Yaskawa INFORM job: A_ROOF_UPPER_0614_2_PAINT_31.JBI

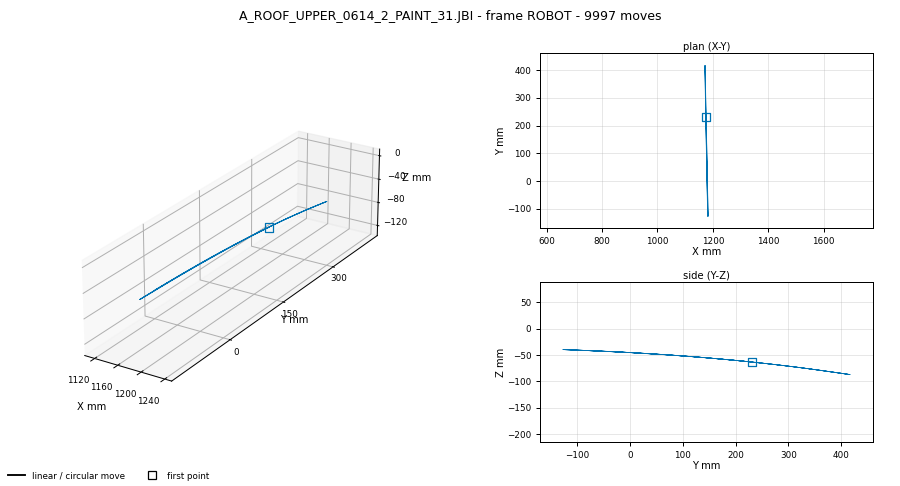
[picture p0: tool path of A_ROOF_UPPER_0614_2_PAINT_31.JBI in frame ROBOT, 9997 of 9997 moves have a stored position in this frame; points joined in program order, loops and branches not executed]
/JOB
//NAME A_ROOF_UPPER_0614_2_PAINT31
//POS
///NPOS 9997,0,0,0,0,0
///TOOL 1
///USER 0
///POSTYPE ROBOT
///RECTAN
///RCONF 1,0,0,0,0,0,0,0,0,0,0,0,0,0,0,0,0,0,0,0,0,0,0,0
C00000=1175.962,231.561,-63.142,-177.522,7.133,148.611
C00001=1175.967,231.312,-63.116,-177.525,7.130,148.612
C00002=1175.971,231.063,-63.091,-177.528,7.128,148.612
C00003=1175.976,230.815,-63.065,-177.530,7.126,148.612
C00004=1175.980,230.567,-63.040,-177.533,7.123,148.612
C00005=1175.985,230.317,-63.013,-177.535,7.121,148.612
C00006=1175.989,230.069,-62.987,-177.539,7.118,148.613
C00007=1175.994,229.820,-62.962,-177.541,7.116,148.613
C00008=1175.998,229.572,-62.936,-177.544,7.113,148.613
C00009=1176.002,229.323,-62.911,-177.546,7.111,148.613
C00010=1176.007,229.075,-62.885,-177.550,7.109,148.614
C00011=1176.011,228.826,-62.859,-177.552,7.107,148.614
C00012=1176.016,228.577,-62.834,-177.555,7.104,148.614
C00013=1176.020,228.328,-62.808,-177.557,7.102,148.614
C00014=1176.025,228.080,-62.783,-177.560,7.099,148.614
C00015=1176.030,227.831,-62.756,-177.563,7.097,148.614
C00016=1176.034,227.582,-62.730,-177.565,7.094,148.615
C00017=1176.039,227.334,-62.705,-177.568,7.092,148.615
C00018=1176.043,227.085,-62.679,-177.571,7.089,148.615
C00019=1176.047,226.837,-62.654,-177.573,7.087,148.615
C00020=1176.052,226.589,-62.628,-177.576,7.085,148.615
C00021=1176.057,226.339,-62.603,-177.579,7.083,148.616
C00022=1176.061,226.091,-62.578,-177.581,7.081,148.616
C00023=1176.066,225.842,-62.552,-177.584,7.078,148.616
C00024=1176.070,225.593,-62.526,-177.586,7.076,148.616
C00025=1176.075,225.345,-62.501,-177.590,7.073,148.616
C00026=1176.079,225.096,-62.476,-177.592,7.071,148.617
C00027=1176.083,224.847,-62.450,-177.595,7.068,148.617
C00028=1176.088,224.599,-62.425,-177.597,7.066,148.617
C00029=1176.092,224.350,-62.400,-177.600,7.065,148.617
C00030=1176.097,224.102,-62.375,-177.603,7.062,148.618
C00031=1176.101,223.853,-62.349,-177.605,7.060,148.618
C00032=1176.105,223.604,-62.323,-177.608,7.057,148.618
C00033=1176.110,223.356,-62.298,-177.611,7.055,148.618
C00034=1176.115,223.107,-62.273,-177.614,7.052,148.618
C00035=1176.119,222.858,-62.248,-177.616,7.050,148.619
C00036=1176.124,222.610,-62.222,-177.619,7.048,148.619
C00037=1176.129,222.361,-62.197,-177.621,7.045,148.619
C00038=1176.133,222.112,-62.171,-177.624,7.044,148.619
C00039=1176.137,221.863,-62.146,-177.627,7.041,148.619
C00040=1176.142,221.615,-62.122,-177.630,7.039,148.620
C00041=1176.146,221.366,-62.096,-177.632,7.036,148.620
C00042=1176.151,221.117,-62.071,-177.635,7.034,148.620
C00043=1176.155,220.869,-62.045,-177.637,7.032,148.620
C00044=1176.160,220.620,-62.020,-177.640,7.029,148.621
C00045=1176.165,220.371,-61.995,-177.643,7.028,148.621
C00046=1176.169,220.123,-61.970,-177.646,7.025,148.621
C00047=1176.173,219.874,-61.945,-177.648,7.023,148.621
C00048=1176.178,219.626,-61.920,-177.651,7.021,148.621
C00049=1176.183,219.376,-61.895,-177.654,7.018,148.622
C00050=1176.187,219.129,-61.870,-177.656,7.016,148.622
C00051=1176.191,218.879,-61.845,-177.659,7.013,148.622
C00052=1176.196,218.631,-61.820,-177.662,7.012,148.623
C00053=1176.201,218.382,-61.795,-177.664,7.009,148.623
C00054=1176.205,218.134,-61.770,-177.667,7.007,148.623
C00055=1176.209,217.884,-61.745,-177.670,7.005,148.623
C00056=1176.214,217.636,-61.720,-177.673,7.002,148.623
C00057=1176.219,217.387,-61.694,-177.675,7.000,148.623
C00058=1176.223,217.138,-61.670,-177.678,6.998,148.624
C00059=1176.227,216.890,-61.644,-177.681,6.996,148.624
C00060=1176.232,216.641,-61.620,-177.683,6.993,148.624
C00061=1176.236,216.392,-61.595,-177.686,6.991,148.625
C00062=1176.241,216.144,-61.570,-177.688,6.989,148.625
C00063=1176.245,215.894,-61.545,-177.691,6.987,148.625
C00064=1176.250,215.646,-61.521,-177.694,6.984,148.625
C00065=1176.255,215.398,-61.495,-177.697,6.982,148.625
C00066=1176.259,215.148,-61.470,-177.699,6.980,148.626
C00067=1176.264,214.900,-61.446,-177.702,6.977,148.626
C00068=1176.268,214.651,-61.421,-177.705,6.976,148.626
C00069=1176.273,214.402,-61.396,-177.708,6.973,148.626
C00070=1176.277,214.153,-61.371,-177.710,6.971,148.627
C00071=1176.282,213.905,-61.347,-177.713,6.969,148.627
C00072=1176.287,213.656,-61.321,-177.715,6.966,148.627
C00073=1176.290,213.407,-61.297,-177.718,6.964,148.627
C00074=1176.296,213.159,-61.272,-177.721,6.962,148.628
C00075=1176.300,212.910,-61.248,-177.724,6.960,148.628
C00076=1176.305,212.661,-61.223,-177.726,6.958,148.628
C00077=1176.309,212.413,-61.198,-177.728,6.956,148.628
C00078=1176.313,212.164,-61.173,-177.732,6.953,148.629
C00079=1176.318,211.915,-61.149,-177.734,6.951,148.629
C00080=1176.323,211.666,-61.125,-177.736,6.949,148.629
C00081=1176.327,211.417,-61.100,-177.740,6.946,148.629
C00082=1176.332,211.169,-61.076,-177.742,6.945,148.630
C00083=1176.337,210.920,-61.051,-177.745,6.942,148.630
C00084=1176.341,210.649,-61.024,-177.748,6.940,148.630
C00085=1176.346,210.379,-60.998,-177.751,6.937,148.630
C00086=1176.351,210.109,-60.971,-177.754,6.935,148.631
C00087=1176.355,209.838,-60.944,-177.756,6.933,148.631
C00088=1176.361,209.589,-60.919,-177.759,6.931,148.631
C00089=1176.365,209.341,-60.895,-177.762,6.928,148.631
C00090=1176.369,209.092,-60.870,-177.765,6.926,148.632
C00091=1176.374,208.843,-60.846,-177.767,6.924,148.632
C00092=1176.379,208.594,-60.821,-177.770,6.922,148.632
C00093=1176.383,208.346,-60.797,-177.773,6.919,148.632
C00094=1176.387,208.097,-60.773,-177.775,6.918,148.633
C00095=1176.392,207.848,-60.748,-177.779,6.915,148.633
C00096=1176.397,207.600,-60.724,-177.781,6.913,148.633
C00097=1176.402,207.351,-60.699,-177.783,6.911,148.634
C00098=1176.406,207.102,-60.675,-177.787,6.909,148.634
C00099=1176.411,206.853,-60.651,-177.789,6.906,148.634
C00100=1176.415,206.604,-60.627,-177.791,6.905,148.634
C00101=1176.420,206.356,-60.603,-177.795,6.902,148.635
C00102=1176.424,206.106,-60.578,-177.797,6.900,148.635
C00103=1176.429,205.858,-60.554,-177.800,6.898,148.635
C00104=1176.433,205.609,-60.530,-177.802,6.896,148.635
C00105=1176.438,205.361,-60.505,-177.805,6.893,148.636
C00106=1176.442,205.111,-60.481,-177.808,6.892,148.636
C00107=1176.447,204.863,-60.457,-177.810,6.890,148.636
C00108=1176.452,204.614,-60.433,-177.813,6.887,148.636
C00109=1176.456,204.365,-60.408,-177.816,6.885,148.637
C00110=1176.461,204.117,-60.384,-177.818,6.883,148.637
C00111=1176.466,203.867,-60.360,-177.821,6.880,148.637
C00112=1176.470,203.619,-60.336,-177.824,6.878,148.637
C00113=1176.474,203.370,-60.312,-177.827,6.877,148.638
C00114=1176.479,203.122,-60.288,-177.829,6.875,148.638
C00115=1176.484,202.872,-60.264,-177.832,6.872,148.638
C00116=1176.488,202.623,-60.239,-177.835,6.870,148.639
C00117=1176.492,202.375,-60.215,-177.837,6.868,148.639
C00118=1176.497,202.126,-60.192,-177.840,6.865,148.639
C00119=1176.502,201.877,-60.167,-177.843,6.864,148.639
C00120=1176.507,201.629,-60.143,-177.845,6.862,148.640
C00121=1176.511,201.380,-60.120,-177.848,6.860,148.640
C00122=1176.515,201.131,-60.096,-177.851,6.857,148.640
C00123=1176.519,200.882,-60.071,-177.853,6.855,148.640
C00124=1176.525,200.633,-60.047,-177.856,6.853,148.641
C00125=1176.529,200.384,-60.023,-177.859,6.851,148.641
C00126=1176.534,200.135,-60.000,-177.862,6.849,148.641
C00127=1176.538,199.887,-59.976,-177.864,6.847,148.642
C00128=1176.543,199.639,-59.952,-177.866,6.845,148.642
C00129=1176.547,199.389,-59.928,-177.870,6.842,148.642
C00130=1176.552,199.140,-59.904,-177.872,6.840,148.642
C00131=1176.557,198.891,-59.880,-177.875,6.839,148.643
C00132=1176.561,198.643,-59.856,-177.877,6.837,148.643
C00133=1176.566,198.394,-59.833,-177.880,6.834,148.643
C00134=1176.570,198.145,-59.809,-177.883,6.832,148.644
C00135=1176.575,197.896,-59.785,-177.885,6.830,148.644
C00136=1176.579,197.648,-59.761,-177.888,6.828,148.644
C00137=1176.584,197.399,-59.738,-177.891,6.826,148.644
C00138=1176.588,197.150,-59.714,-177.894,6.824,148.645
C00139=1176.593,196.901,-59.690,-177.896,6.822,148.645
C00140=1176.598,196.653,-59.666,-177.899,6.820,148.645
C00141=1176.602,196.403,-59.642,-177.902,6.817,148.646
C00142=1176.607,196.154,-59.619,-177.905,6.816,148.646
C00143=1176.611,195.905,-59.595,-177.907,6.813,148.646
C00144=1176.616,195.656,-59.571,-177.910,6.812,148.646
C00145=1176.621,195.407,-59.548,-177.913,6.809,148.647
C00146=1176.625,195.159,-59.524,-177.915,6.807,148.647
C00147=1176.630,194.910,-59.500,-177.918,6.805,148.647
C00148=1176.635,194.661,-59.477,-177.920,6.803,148.648
C00149=1176.639,194.412,-59.453,-177.923,6.802,148.648
C00150=1176.644,194.163,-59.430,-177.926,6.799,148.648
C00151=1176.648,193.914,-59.406,-177.928,6.797,148.648
C00152=1176.653,193.666,-59.382,-177.931,6.795,148.649
C00153=1176.657,193.417,-59.359,-177.934,6.793,148.649
C00154=1176.662,193.168,-59.335,-177.937,6.791,148.649
C00155=1176.667,192.919,-59.312,-177.940,6.789,148.650
C00156=1176.671,192.670,-59.288,-177.942,6.787,148.650
C00157=1176.675,192.422,-59.265,-177.945,6.785,148.650
C00158=1176.680,192.173,-59.242,-177.947,6.783,148.651
C00159=1176.685,191.924,-59.219,-177.950,6.781,148.651
C00160=1176.689,191.675,-59.195,-177.953,6.779,148.651
C00161=1176.694,191.426,-59.171,-177.955,6.777,148.651
C00162=1176.699,191.178,-59.148,-177.958,6.775,148.652
C00163=1176.704,190.929,-59.125,-177.961,6.773,148.652
C00164=1176.708,190.680,-59.101,-177.964,6.771,148.652
C00165=1176.713,190.431,-59.078,-177.966,6.768,148.652
C00166=1176.718,190.182,-59.055,-177.969,6.767,148.653
C00167=1176.721,189.934,-59.031,-177.971,6.765,148.653
C00168=1176.726,189.685,-59.008,-177.974,6.763,148.654
C00169=1176.731,189.436,-58.985,-177.977,6.760,148.654
C00170=1176.736,189.187,-58.961,-177.980,6.758,148.654
C00171=1176.740,188.938,-58.938,-177.982,6.757,148.654
C00172=1176.745,188.688,-58.914,-177.985,6.755,148.655
C00173=1176.749,188.440,-58.892,-177.988,6.753,148.655
C00174=1176.754,188.191,-58.869,-177.991,6.750,148.655
C00175=1176.759,187.942,-58.845,-177.993,6.748,148.656
C00176=1176.764,187.693,-58.822,-177.996,6.747,148.656
C00177=1176.768,187.444,-58.799,-177.998,6.745,148.656
C00178=1176.772,187.196,-58.776,-178.001,6.743,148.657
C00179=1176.777,186.947,-58.752,-178.004,6.741,148.657
C00180=1176.782,186.698,-58.729,-178.007,6.739,148.657
C00181=1176.786,186.449,-58.706,-178.009,6.736,148.657
C00182=1176.791,186.200,-58.683,-178.012,6.735,148.658
C00183=1176.796,185.951,-58.660,-178.014,6.733,148.658
C00184=1176.800,185.702,-58.637,-178.017,6.731,148.659
C00185=1176.805,185.453,-58.613,-178.020,6.729,148.659
C00186=1176.809,185.204,-58.591,-178.023,6.727,148.659
C00187=1176.814,184.955,-58.568,-178.025,6.725,148.659
C00188=1176.819,184.685,-58.543,-178.028,6.723,148.660
C00189=1176.824,184.416,-58.518,-178.031,6.720,148.660
C00190=1176.829,184.147,-58.493,-178.034,6.718,148.660
C00191=1176.834,183.877,-58.468,-178.037,6.716,148.661
C00192=1176.838,183.628,-58.445,-178.040,6.714,148.661
C00193=1176.844,183.379,-58.423,-178.042,6.712,148.661
C00194=1176.848,183.131,-58.400,-178.045,6.711,148.662
C00195=1176.852,182.881,-58.376,-178.048,6.709,148.662
C00196=1176.857,182.632,-58.353,-178.051,6.707,148.662
C00197=1176.862,182.384,-58.331,-178.053,6.705,148.663
C00198=1176.867,182.135,-58.308,-178.056,6.702,148.663
C00199=1176.871,181.886,-58.285,-178.059,6.701,148.663
C00200=1176.875,181.637,-58.262,-178.061,6.699,148.664
C00201=1176.880,181.387,-58.239,-178.064,6.697,148.664
C00202=1176.885,181.139,-58.217,-178.067,6.695,148.664
C00203=1176.890,180.890,-58.194,-178.069,6.693,148.665
C00204=1176.894,180.642,-58.171,-178.072,6.691,148.665
C00205=1176.899,180.392,-58.148,-178.074,6.690,148.665
C00206=1176.904,180.144,-58.125,-178.077,6.687,148.666
C00207=1176.908,179.895,-58.102,-178.080,6.685,148.666
C00208=1176.913,179.645,-58.080,-178.083,6.683,148.666
C00209=1176.917,179.397,-58.057,-178.085,6.682,148.667
C00210=1176.923,179.148,-58.035,-178.088,6.680,148.667
C00211=1176.926,178.899,-58.012,-178.091,6.678,148.667
C00212=1176.931,178.650,-57.989,-178.093,6.676,148.668
C00213=1176.936,178.401,-57.967,-178.096,6.674,148.668
C00214=1176.941,178.152,-57.944,-178.099,6.672,148.668
C00215=1176.945,177.903,-57.921,-178.102,6.670,148.669
C00216=1176.950,177.654,-57.898,-178.104,6.668,148.669
C00217=1176.955,177.405,-57.876,-178.107,6.666,148.669
C00218=1176.959,177.156,-57.853,-178.110,6.664,148.670
C00219=1176.964,176.907,-57.831,-178.112,6.663,148.670
C00220=1176.968,176.659,-57.809,-178.115,6.661,148.670
C00221=1176.973,176.409,-57.786,-178.117,6.659,148.671
C00222=1176.977,176.160,-57.763,-178.120,6.657,148.671
C00223=1176.983,175.911,-57.741,-178.123,6.655,148.671
C00224=1176.987,175.663,-57.718,-178.126,6.653,148.672
C00225=1176.992,175.414,-57.696,-178.129,6.651,148.672
C00226=1176.996,175.165,-57.673,-178.131,6.649,148.672
C00227=1177.000,174.916,-57.651,-178.134,6.647,148.673
C00228=1177.006,174.667,-57.628,-178.137,6.646,148.673
C00229=1177.010,174.418,-57.606,-178.139,6.644,148.673
C00230=1177.014,174.169,-57.584,-178.142,6.642,148.674
C00231=1177.020,173.920,-57.561,-178.145,6.640,148.674
C00232=1177.024,173.671,-57.539,-178.147,6.638,148.674
C00233=1177.029,173.422,-57.517,-178.149,6.636,148.675
C00234=1177.033,173.173,-57.494,-178.152,6.635,148.675
C00235=1177.038,172.924,-57.472,-178.155,6.632,148.675
C00236=1177.043,172.675,-57.450,-178.158,6.630,148.676
C00237=1177.047,172.426,-57.427,-178.161,6.628,148.676
C00238=1177.052,172.178,-57.405,-178.163,6.627,148.676
C00239=1177.056,171.928,-57.383,-178.166,6.625,148.677
C00240=1177.061,171.679,-57.360,-178.169,6.623,148.677
C00241=1177.066,171.431,-57.338,-178.172,6.621,148.678
C00242=1177.070,171.181,-57.316,-178.174,6.620,148.678
C00243=1177.076,170.932,-57.294,-178.177,6.618,148.678
C00244=1177.080,170.684,-57.271,-178.180,6.616,148.679
C00245=1177.085,170.435,-57.249,-178.182,6.614,148.679
C00246=1177.089,170.186,-57.227,-178.184,6.612,148.679
C00247=1177.095,169.937,-57.205,-178.187,6.610,148.680
C00248=1177.099,169.687,-57.183,-178.190,6.609,148.680
C00249=1177.103,169.439,-57.161,-178.192,6.607,148.680
C00250=1177.108,169.190,-57.138,-178.195,6.605,148.681
C00251=1177.113,168.940,-57.116,-178.198,6.603,148.681
C00252=1177.118,168.692,-57.094,-178.201,6.601,148.681
C00253=1177.122,168.442,-57.072,-178.204,6.599,148.682
C00254=1177.127,168.194,-57.050,-178.206,6.597,148.682
C00255=1177.131,167.944,-57.028,-178.209,6.595,148.682
C00256=1177.137,167.695,-57.006,-178.212,6.594,148.683
C00257=1177.141,167.447,-56.983,-178.215,6.592,148.683
C00258=1177.145,167.198,-56.962,-178.217,6.590,148.684
C00259=1177.150,166.949,-56.940,-178.220,6.588,148.684
C00260=1177.155,166.700,-56.918,-178.223,6.587,148.684
C00261=1177.159,166.451,-56.896,-178.225,6.585,148.685
C00262=1177.164,166.202,-56.874,-178.228,6.583,148.685
C00263=1177.169,165.953,-56.852,-178.231,6.581,148.685
C00264=1177.174,165.704,-56.830,-178.233,6.580,148.686
C00265=1177.178,165.455,-56.808,-178.236,6.578,148.686
C00266=1177.183,165.206,-56.786,-178.239,6.576,148.687
C00267=1177.188,164.957,-56.764,-178.241,6.574,148.687
C00268=1177.192,164.708,-56.742,-178.244,6.572,148.687
C00269=1177.197,164.459,-56.721,-178.247,6.571,148.688
C00270=1177.201,164.210,-56.699,-178.249,6.569,148.688
C00271=1177.206,163.961,-56.677,-178.252,6.567,148.688
C00272=1177.211,163.713,-56.655,-178.255,6.565,148.689
C00273=1177.215,163.463,-56.634,-178.257,6.564,148.689
C00274=1177.220,163.214,-56.612,-178.260,6.562,148.689
C00275=1177.224,162.965,-56.590,-178.263,6.560,148.690
C00276=1177.229,162.716,-56.569,-178.266,6.558,148.690
C00277=1177.234,162.467,-56.547,-178.268,6.557,148.691
C00278=1177.238,162.218,-56.525,-178.271,6.555,148.691
C00279=1177.243,161.969,-56.503,-178.274,6.553,148.691
C00280=1177.248,161.719,-56.482,-178.276,6.551,148.692
C00281=1177.253,161.471,-56.460,-178.279,6.550,148.692
C00282=1177.258,161.222,-56.438,-178.282,6.548,148.692
C00283=1177.262,160.973,-56.416,-178.284,6.546,148.693
C00284=1177.267,160.724,-56.395,-178.287,6.544,148.693
C00285=1177.272,160.475,-56.374,-178.290,6.542,148.694
C00286=1177.276,160.226,-56.352,-178.292,6.541,148.694
C00287=1177.281,159.977,-56.330,-178.295,6.539,148.694
C00288=1177.285,159.728,-56.308,-178.298,6.537,148.695
C00289=1177.290,159.478,-56.287,-178.300,6.535,148.695
C00290=1177.295,159.230,-56.265,-178.303,6.534,148.695
C00291=1177.300,158.980,-56.243,-178.306,6.532,148.696
C00292=1177.305,158.712,-56.221,-178.309,6.530,148.696
C00293=1177.310,158.443,-56.198,-178.311,6.528,148.697
C00294=1177.315,158.174,-56.174,-178.314,6.526,148.697
C00295=1177.320,157.905,-56.151,-178.317,6.524,148.697
C00296=1177.325,157.655,-56.129,-178.320,6.522,148.698
C00297=1177.330,157.406,-56.108,-178.323,6.521,148.698
C00298=1177.334,157.158,-56.087,-178.326,6.519,148.699
C00299=1177.339,156.909,-56.065,-178.328,6.517,148.699
C00300=1177.343,156.659,-56.044,-178.331,6.516,148.699
C00301=1177.348,156.411,-56.022,-178.334,6.514,148.700
C00302=1177.353,156.161,-56.001,-178.336,6.512,148.700
C00303=1177.358,155.912,-55.979,-178.339,6.510,148.701
C00304=1177.362,155.663,-55.958,-178.342,6.509,148.701
C00305=1177.367,155.414,-55.937,-178.344,6.508,148.701
C00306=1177.372,155.166,-55.915,-178.347,6.506,148.702
C00307=1177.376,154.916,-55.894,-178.349,6.504,148.702
C00308=1177.381,154.667,-55.872,-178.352,6.502,148.702
C00309=1177.386,154.418,-55.852,-178.355,6.501,148.703
C00310=1177.391,154.170,-55.830,-178.357,6.499,148.703
C00311=1177.395,153.920,-55.809,-178.360,6.497,148.704
C00312=1177.400,153.671,-55.787,-178.363,6.495,148.704
C00313=1177.405,153.422,-55.767,-178.365,6.494,148.704
C00314=1177.410,153.173,-55.746,-178.368,6.492,148.705
C00315=1177.415,152.924,-55.724,-178.371,6.490,148.705
C00316=1177.419,152.674,-55.703,-178.374,6.488,148.705
C00317=1177.423,152.426,-55.682,-178.377,6.487,148.706
C00318=1177.428,152.177,-55.661,-178.379,6.485,148.706
C00319=1177.433,151.928,-55.639,-178.382,6.483,148.707
C00320=1177.438,151.679,-55.619,-178.385,6.482,148.707
C00321=1177.442,151.429,-55.597,-178.387,6.481,148.708
C00322=1177.447,151.180,-55.576,-178.390,6.479,148.708
C00323=1177.452,150.931,-55.555,-178.392,6.477,148.708
C00324=1177.457,150.682,-55.534,-178.395,6.475,148.709
C00325=1177.462,150.434,-55.513,-178.398,6.474,148.709
C00326=1177.466,150.184,-55.491,-178.400,6.472,148.709
C00327=1177.471,149.935,-55.471,-178.403,6.470,148.710
C00328=1177.476,149.686,-55.449,-178.406,6.468,148.710
C00329=1177.480,149.437,-55.429,-178.408,6.467,148.711
C00330=1177.485,149.188,-55.408,-178.412,6.465,148.711
C00331=1177.490,148.939,-55.387,-178.414,6.463,148.712
C00332=1177.494,148.690,-55.366,-178.417,6.462,148.712
C00333=1177.499,148.440,-55.344,-178.419,6.461,148.712
C00334=1177.503,148.191,-55.324,-178.422,6.459,148.713
C00335=1177.509,147.942,-55.303,-178.424,6.457,148.713
C00336=1177.514,147.693,-55.281,-178.427,6.455,148.713
C00337=1177.518,147.445,-55.261,-178.430,6.454,148.714
C00338=1177.523,147.195,-55.240,-178.433,6.452,148.714
C00339=1177.528,146.946,-55.220,-178.435,6.450,148.715
C00340=1177.533,146.697,-55.199,-178.438,6.449,148.715
C00341=1177.537,146.449,-55.178,-178.441,6.447,148.716
C00342=1177.541,146.199,-55.156,-178.444,6.445,148.716
C00343=1177.547,145.949,-55.135,-178.446,6.444,148.716
C00344=1177.551,145.701,-55.115,-178.449,6.443,148.717
C00345=1177.556,145.451,-55.094,-178.451,6.441,148.717
C00346=1177.561,145.202,-55.074,-178.454,6.439,148.718
C00347=1177.566,144.953,-55.053,-178.457,6.437,148.718
C00348=1177.570,144.704,-55.032,-178.459,6.436,148.718
C00349=1177.575,144.455,-55.011,-178.463,6.434,148.719
C00350=1177.580,144.207,-54.990,-178.465,6.432,148.719
C00351=1177.584,143.958,-54.970,-178.467,6.432,148.720
C00352=1177.589,143.708,-54.949,-178.470,6.430,148.720
C00353=1177.594,143.459,-54.929,-178.473,6.428,148.720
C00354=1177.599,143.210,-54.908,-178.475,6.426,148.721
C00355=1177.603,142.961,-54.887,-178.478,6.425,148.721
C00356=1177.608,142.712,-54.866,-178.481,6.423,148.722
C00357=1177.613,142.463,-54.846,-178.484,6.421,148.722
C00358=1177.617,142.214,-54.825,-178.487,6.420,148.723
C00359=1177.622,141.965,-54.805,-178.489,6.419,148.723
C00360=1177.627,141.716,-54.784,-178.492,6.417,148.723
C00361=1177.632,141.467,-54.763,-178.494,6.415,148.724
C00362=1177.637,141.217,-54.744,-178.497,6.413,148.724
C00363=1177.641,140.968,-54.723,-178.500,6.412,148.725
C00364=1177.646,140.719,-54.702,-178.502,6.410,148.725
C00365=1177.651,140.470,-54.682,-178.505,6.409,148.726
C00366=1177.656,140.221,-54.661,-178.508,6.408,148.726
C00367=1177.660,139.972,-54.640,-178.510,6.406,148.726
C00368=1177.665,139.723,-54.620,-178.513,6.404,148.727
C00369=1177.670,139.473,-54.599,-178.516,6.402,148.727
C00370=1177.675,139.224,-54.579,-178.518,6.401,148.728
C00371=1177.679,138.975,-54.559,-178.522,6.399,148.728
C00372=1177.684,138.726,-54.538,-178.524,6.398,148.729
C00373=1177.689,138.477,-54.518,-178.526,6.397,148.729
C00374=1177.693,138.228,-54.497,-178.529,6.395,148.729
C00375=1177.698,137.979,-54.477,-178.532,6.393,148.730
C00376=1177.703,137.729,-54.457,-178.534,6.391,148.730
C00377=1177.708,137.480,-54.436,-178.538,6.390,148.731
C00378=1177.712,137.231,-54.416,-178.540,6.389,148.731
C00379=1177.717,136.982,-54.395,-178.542,6.387,148.731
C00380=1177.722,136.733,-54.375,-178.545,6.385,148.732
C00381=1177.726,136.483,-54.355,-178.548,6.384,148.732
C00382=1177.732,136.235,-54.335,-178.551,6.382,148.733
C00383=1177.736,135.986,-54.315,-178.554,6.381,148.733
C00384=1177.741,135.736,-54.294,-178.556,6.380,148.734
C00385=1177.746,135.487,-54.274,-178.559,6.378,148.734
C00386=1177.750,135.238,-54.254,-178.561,6.376,148.734
C00387=1177.755,134.989,-54.234,-178.564,6.374,148.735
C00388=1177.760,134.739,-54.213,-178.567,6.373,148.735
C00389=1177.765,134.490,-54.193,-178.569,6.372,148.736
C00390=1177.769,134.241,-54.173,-178.572,6.370,148.736
C00391=1177.774,133.993,-54.153,-178.575,6.369,148.737
C00392=1177.779,133.744,-54.133,-178.577,6.367,148.737
C00393=1177.784,133.494,-54.113,-178.580,6.365,148.737
C00394=1177.789,133.245,-54.092,-178.583,6.364,148.738
C00395=1177.794,132.995,-54.072,-178.585,6.363,148.738
C00396=1177.798,132.727,-54.051,-178.588,6.361,148.739
C00397=1177.804,132.458,-54.029,-178.591,6.359,148.739
C00398=1177.808,132.190,-54.007,-178.594,6.358,148.740
C00399=1177.814,131.921,-53.985,-178.597,6.356,148.740
C00400=1177.819,131.672,-53.966,-178.599,6.354,148.741
C00401=1177.823,131.423,-53.945,-178.602,6.353,148.741
C00402=1177.829,131.174,-53.926,-178.605,6.351,148.742
C00403=1177.833,130.925,-53.906,-178.607,6.350,148.742
C00404=1177.838,130.675,-53.886,-178.610,6.349,148.742
C00405=1177.842,130.426,-53.866,-178.613,6.347,148.743
C00406=1177.847,130.177,-53.846,-178.616,6.345,148.743
C00407=1177.852,129.929,-53.826,-178.619,6.344,148.744
C00408=1177.857,129.679,-53.806,-178.621,6.343,148.744
C00409=1177.862,129.430,-53.785,-178.623,6.341,148.745
C00410=1177.867,129.180,-53.766,-178.626,6.339,148.745
C00411=1177.872,128.931,-53.746,-178.629,6.338,148.746
C00412=1177.876,128.682,-53.726,-178.631,6.337,148.746
C00413=1177.881,128.433,-53.706,-178.634,6.335,148.746
C00414=1177.886,128.184,-53.686,-178.637,6.333,148.747
C00415=1177.891,127.935,-53.667,-178.640,6.332,148.747
C00416=1177.896,127.685,-53.647,-178.642,6.331,148.748
C00417=1177.900,127.437,-53.627,-178.645,6.329,148.748
C00418=1177.905,127.187,-53.607,-178.648,6.328,148.749
C00419=1177.910,126.938,-53.588,-178.650,6.326,148.749
C00420=1177.915,126.689,-53.567,-178.653,6.325,148.750
C00421=1177.919,126.440,-53.548,-178.656,6.324,148.750
C00422=1177.923,126.190,-53.529,-178.658,6.322,148.750
C00423=1177.928,125.942,-53.509,-178.661,6.320,148.751
C00424=1177.933,125.693,-53.489,-178.664,6.320,148.751
C00425=1177.938,125.443,-53.469,-178.666,6.318,148.752
C00426=1177.943,125.193,-53.450,-178.669,6.316,148.752
C00427=1177.948,124.945,-53.430,-178.672,6.314,148.753
C00428=1177.952,124.696,-53.410,-178.674,6.314,148.753
C00429=1177.957,124.446,-53.390,-178.677,6.312,148.754
C00430=1177.963,124.197,-53.371,-178.680,6.310,148.754
C00431=1177.967,123.948,-53.351,-178.682,6.309,148.754
C00432=1177.972,123.699,-53.331,-178.685,6.308,148.755
C00433=1177.976,123.450,-53.312,-178.688,6.306,148.755
C00434=1177.981,123.200,-53.293,-178.690,6.305,148.756
C00435=1177.986,122.951,-53.273,-178.693,6.303,148.756
C00436=1177.991,122.703,-53.253,-178.696,6.302,148.757
C00437=1177.996,122.453,-53.233,-178.698,6.300,148.757
C00438=1178.000,122.204,-53.214,-178.701,6.299,148.758
C00439=1178.006,121.955,-53.194,-178.704,6.297,148.758
C00440=1178.010,121.705,-53.175,-178.706,6.296,148.759
C00441=1178.014,121.456,-53.156,-178.709,6.295,148.759
C00442=1178.020,121.207,-53.136,-178.712,6.293,148.760
C00443=1178.025,120.957,-53.117,-178.714,6.292,148.760
C00444=1178.030,120.709,-53.097,-178.717,6.291,148.761
C00445=1178.034,120.459,-53.078,-178.720,6.289,148.761
C00446=1178.039,120.210,-53.059,-178.723,6.287,148.761
C00447=1178.044,119.961,-53.039,-178.725,6.286,148.762
C00448=1178.048,119.712,-53.019,-178.728,6.285,148.762
C00449=1178.054,119.463,-53.000,-178.731,6.283,148.763
C00450=1178.058,119.214,-52.981,-178.733,6.282,148.763
C00451=1178.062,118.964,-52.961,-178.736,6.281,148.764
C00452=1178.068,118.715,-52.942,-178.739,6.279,148.764
C00453=1178.073,118.466,-52.922,-178.741,6.278,148.765
C00454=1178.077,118.217,-52.903,-178.743,6.276,148.765
C00455=1178.082,117.967,-52.885,-178.747,6.275,148.766
C00456=1178.087,117.717,-52.865,-178.749,6.273,148.766
C00457=1178.092,117.469,-52.846,-178.751,6.272,148.766
C00458=1178.096,117.219,-52.827,-178.755,6.271,148.767
C00459=1178.102,116.970,-52.807,-178.757,6.269,148.768
C00460=1178.106,116.721,-52.788,-178.760,6.268,148.768
C00461=1178.111,116.472,-52.769,-178.762,6.267,148.768
C00462=1178.116,116.223,-52.749,-178.765,6.265,148.769
C00463=1178.121,115.974,-52.730,-178.768,6.264,148.769
C00464=1178.125,115.725,-52.711,-178.770,6.263,148.770
C00465=1178.131,115.475,-52.692,-178.773,6.261,148.770
C00466=1178.135,115.226,-52.673,-178.776,6.260,148.771
C00467=1178.140,114.977,-52.654,-178.778,6.259,148.771
C00468=1178.145,114.727,-52.634,-178.781,6.257,148.772
C00469=1178.149,114.479,-52.616,-178.784,6.256,148.772
C00470=1178.154,114.229,-52.596,-178.786,6.255,148.773
C00471=1178.160,113.980,-52.577,-178.789,6.253,148.773
C00472=1178.164,113.731,-52.558,-178.792,6.252,148.774
C00473=1178.169,113.482,-52.539,-178.794,6.251,148.774
C00474=1178.173,113.232,-52.520,-178.797,6.249,148.774
C00475=1178.179,112.983,-52.501,-178.800,6.248,148.775
C00476=1178.184,112.733,-52.482,-178.802,6.247,148.776
C00477=1178.188,112.485,-52.463,-178.805,6.245,148.776
C00478=1178.193,112.235,-52.443,-178.808,6.244,148.777
C00479=1178.198,111.986,-52.425,-178.810,6.242,148.777
C00480=1178.203,111.737,-52.406,-178.813,6.241,148.777
C00481=1178.207,111.488,-52.387,-178.815,6.240,148.778
C00482=1178.212,111.238,-52.368,-178.818,6.238,148.778
C00483=1178.217,110.989,-52.349,-178.821,6.237,148.779
C00484=1178.222,110.740,-52.330,-178.823,6.236,148.779
C00485=1178.227,110.490,-52.311,-178.826,6.234,148.780
C00486=1178.232,110.242,-52.292,-178.829,6.233,148.780
C00487=1178.237,109.992,-52.273,-178.831,6.232,148.781
C00488=1178.242,109.743,-52.255,-178.834,6.230,148.781
C00489=1178.246,109.494,-52.236,-178.837,6.229,148.782
C00490=1178.251,109.245,-52.216,-178.839,6.228,148.782
C00491=1178.256,108.996,-52.198,-178.843,6.226,148.783
C00492=1178.261,108.746,-52.179,-178.845,6.226,148.783
C00493=1178.265,108.497,-52.161,-178.847,6.224,148.784
C00494=1178.270,108.247,-52.141,-178.851,6.222,148.784
C00495=1178.275,107.998,-52.123,-178.853,6.221,148.785
C00496=1178.280,107.749,-52.104,-178.855,6.220,148.785
C00497=1178.285,107.499,-52.086,-178.859,6.218,148.786
C00498=1178.290,107.250,-52.066,-178.861,6.217,148.786
C00499=1178.294,107.001,-52.047,-178.863,6.216,148.787
C00500=1178.300,106.733,-52.027,-178.867,6.214,148.787
C00501=1178.305,106.464,-52.008,-178.869,6.213,148.788
C00502=1178.310,106.196,-51.987,-178.872,6.212,148.788
C00503=1178.315,105.928,-51.967,-178.875,6.211,148.789
C00504=1178.320,105.679,-51.948,-178.878,6.209,148.789
C00505=1178.325,105.429,-51.930,-178.880,6.208,148.790
C00506=1178.330,105.180,-51.912,-178.883,6.207,148.790
C00507=1178.335,104.931,-51.892,-178.886,6.205,148.791
C00508=1178.339,104.681,-51.874,-178.888,6.204,148.791
C00509=1178.344,104.432,-51.855,-178.891,6.203,148.792
C00510=1178.349,104.183,-51.837,-178.893,6.202,148.792
C00511=1178.354,103.934,-51.819,-178.896,6.200,148.793
C00512=1178.358,103.684,-51.800,-178.899,6.199,148.793
C00513=1178.364,103.435,-51.781,-178.901,6.198,148.794
C00514=1178.369,103.186,-51.762,-178.904,6.196,148.794
C00515=1178.373,102.936,-51.744,-178.907,6.196,148.795
C00516=1178.379,102.687,-51.726,-178.909,6.194,148.795
C00517=1178.383,102.438,-51.707,-178.913,6.192,148.796
C00518=1178.388,102.189,-51.689,-178.915,6.192,148.796
C00519=1178.392,101.939,-51.671,-178.917,6.190,148.797
C00520=1178.398,101.690,-51.652,-178.920,6.189,148.797
C00521=1178.403,101.441,-51.633,-178.923,6.188,148.798
C00522=1178.407,101.191,-51.615,-178.926,6.186,148.798
C00523=1178.412,100.942,-51.597,-178.928,6.185,148.799
C00524=1178.417,100.693,-51.578,-178.931,6.184,148.799
C00525=1178.422,100.444,-51.560,-178.933,6.183,148.800
C00526=1178.426,100.194,-51.541,-178.936,6.181,148.800
C00527=1178.431,99.945,-51.523,-178.938,6.180,148.801
C00528=1178.437,99.696,-51.505,-178.942,6.179,148.801
C00529=1178.442,99.447,-51.486,-178.944,6.177,148.802
C00530=1178.446,99.197,-51.468,-178.946,6.176,148.802
C00531=1178.451,98.948,-51.450,-178.950,6.175,148.803
C00532=1178.456,98.699,-51.432,-178.952,6.174,148.803
C00533=1178.461,98.449,-51.413,-178.955,6.173,148.804
C00534=1178.465,98.200,-51.394,-178.957,6.172,148.804
C00535=1178.470,97.951,-51.376,-178.960,6.170,148.805
C00536=1178.475,97.702,-51.358,-178.963,6.169,148.805
C00537=1178.480,97.453,-51.340,-178.965,6.168,148.806
C00538=1178.485,97.203,-51.322,-178.968,6.166,148.806
C00539=1178.489,96.954,-51.304,-178.970,6.166,148.807
C00540=1178.495,96.704,-51.285,-178.973,6.164,148.807
C00541=1178.500,96.455,-51.267,-178.976,6.163,148.808
C00542=1178.505,96.206,-51.249,-178.978,6.162,148.808
C00543=1178.509,95.957,-51.231,-178.981,6.161,148.809
C00544=1178.514,95.707,-51.212,-178.984,6.159,148.809
C00545=1178.519,95.458,-51.194,-178.987,6.158,148.810
C00546=1178.524,95.209,-51.176,-178.989,6.157,148.810
C00547=1178.529,94.960,-51.158,-178.992,6.155,148.811
C00548=1178.533,94.711,-51.140,-178.995,6.155,148.811
C00549=1178.539,94.461,-51.122,-178.997,6.153,148.812
C00550=1178.544,94.212,-51.104,-178.999,6.152,148.812
C00551=1178.548,93.962,-51.085,-179.003,6.151,148.813
C00552=1178.553,93.713,-51.068,-179.005,6.150,148.813
C00553=1178.558,93.464,-51.050,-179.008,6.149,148.814
C00554=1178.563,93.215,-51.032,-179.010,6.148,148.814
C00555=1178.568,92.965,-51.014,-179.013,6.146,148.815
C00556=1178.573,92.716,-50.996,-179.015,6.145,148.815
C00557=1178.578,92.466,-50.978,-179.018,6.144,148.816
C00558=1178.582,92.217,-50.960,-179.021,6.142,148.816
C00559=1178.587,91.967,-50.942,-179.023,6.141,148.817
C00560=1178.592,91.718,-50.924,-179.026,6.140,148.817
C00561=1178.597,91.469,-50.906,-179.029,6.139,148.818
C00562=1178.602,91.220,-50.888,-179.031,6.137,148.818
C00563=1178.607,90.971,-50.870,-179.034,6.137,148.819
C00564=1178.612,90.721,-50.852,-179.037,6.135,148.819
C00565=1178.617,90.472,-50.834,-179.039,6.135,148.820
C00566=1178.622,90.222,-50.817,-179.042,6.133,148.820
C00567=1178.627,89.973,-50.799,-179.044,6.132,148.821
C00568=1178.632,89.724,-50.781,-179.048,6.131,148.821
C00569=1178.636,89.475,-50.764,-179.050,6.130,148.822
C00570=1178.640,89.225,-50.745,-179.053,6.128,148.823
C00571=1178.645,88.976,-50.727,-179.055,6.127,148.823
C00572=1178.650,88.726,-50.710,-179.058,6.126,148.824
C00573=1178.655,88.477,-50.692,-179.060,6.125,148.824
C00574=1178.660,88.228,-50.674,-179.063,6.123,148.824
C00575=1178.665,87.979,-50.656,-179.066,6.123,148.825
C00576=1178.670,87.729,-50.639,-179.068,6.121,148.826
C00577=1178.675,87.480,-50.621,-179.071,6.121,148.826
C00578=1178.680,87.231,-50.603,-179.074,6.119,148.827
C00579=1178.684,86.982,-50.585,-179.076,6.118,148.827
C00580=1178.690,86.732,-50.568,-179.079,6.117,148.828
C00581=1178.695,86.483,-50.550,-179.082,6.116,148.828
C00582=1178.699,86.234,-50.532,-179.084,6.114,148.829
C00583=1178.705,85.984,-50.515,-179.087,6.114,148.829
C00584=1178.710,85.735,-50.497,-179.090,6.112,148.830
C00585=1178.714,85.486,-50.479,-179.092,6.111,148.830
C00586=1178.719,85.236,-50.462,-179.095,6.110,148.831
C00587=1178.724,84.987,-50.444,-179.097,6.109,148.831
C00588=1178.729,84.738,-50.426,-179.100,6.108,148.832
C00589=1178.734,84.488,-50.409,-179.103,6.107,148.832
C00590=1178.739,84.239,-50.391,-179.106,6.105,148.833
C00591=1178.743,83.989,-50.374,-179.108,6.105,148.833
C00592=1178.748,83.740,-50.356,-179.111,6.104,148.834
C00593=1178.753,83.491,-50.338,-179.113,6.102,148.835
C00594=1178.758,83.241,-50.321,-179.115,6.101,148.835
C00595=1178.763,82.992,-50.304,-179.119,6.100,148.836
C00596=1178.768,82.742,-50.287,-179.121,6.099,148.836
C00597=1178.773,82.493,-50.269,-179.124,6.098,148.837
C00598=1178.779,82.244,-50.252,-179.126,6.097,148.837
C00599=1178.783,81.995,-50.234,-179.129,6.096,148.838
C00600=1178.788,81.746,-50.217,-179.131,6.095,148.838
C00601=1178.793,81.496,-50.199,-179.135,6.093,148.839
C00602=1178.798,81.247,-50.182,-179.137,6.092,148.839
C00603=1178.802,80.998,-50.164,-179.140,6.091,148.840
C00604=1178.808,80.729,-50.146,-179.142,6.090,148.840
C00605=1178.813,80.461,-50.126,-179.145,6.089,148.841
C00606=1178.819,80.192,-50.108,-179.148,6.088,148.842
C00607=1178.823,79.924,-50.090,-179.151,6.087,148.842
C00608=1178.828,79.675,-50.072,-179.154,6.085,148.843
C00609=1178.833,79.425,-50.055,-179.156,6.084,148.843
C00610=1178.838,79.175,-50.038,-179.159,6.084,148.844
C00611=1178.843,78.927,-50.020,-179.161,6.082,148.844
C00612=1178.849,78.677,-50.003,-179.164,6.082,148.845
C00613=1178.853,78.428,-49.986,-179.167,6.080,148.845
C00614=1178.858,78.178,-49.968,-179.169,6.079,148.846
C00615=1178.863,77.929,-49.951,-179.172,6.078,148.846
C00616=1178.867,77.680,-49.934,-179.175,6.077,148.847
C00617=1178.873,77.430,-49.916,-179.177,6.076,148.847
C00618=1178.877,77.181,-49.900,-179.180,6.075,148.848
C00619=1178.883,76.932,-49.882,-179.182,6.074,148.849
C00620=1178.888,76.682,-49.865,-179.185,6.072,148.849
C00621=1178.892,76.433,-49.848,-179.188,6.072,148.850
C00622=1178.897,76.184,-49.830,-179.190,6.070,148.850
C00623=1178.902,75.934,-49.814,-179.193,6.070,148.851
C00624=1178.907,75.684,-49.796,-179.195,6.069,148.851
C00625=1178.912,75.436,-49.779,-179.198,6.067,148.852
C00626=1178.917,75.186,-49.762,-179.200,6.066,148.852
C00627=1178.922,74.937,-49.745,-179.204,6.065,148.853
C00628=1178.927,74.687,-49.728,-179.206,6.064,148.853
C00629=1178.932,74.438,-49.710,-179.209,6.063,148.854
C00630=1178.937,74.189,-49.694,-179.211,6.062,148.854
C00631=1178.942,73.939,-49.677,-179.214,6.061,148.855
C00632=1178.946,73.690,-49.660,-179.217,6.060,148.855
C00633=1178.952,73.440,-49.643,-179.219,6.059,148.856
C00634=1178.956,73.191,-49.625,-179.222,6.057,148.857
C00635=1178.962,72.942,-49.608,-179.225,6.057,148.857
C00636=1178.966,72.693,-49.592,-179.227,6.056,148.858
C00637=1178.971,72.443,-49.574,-179.230,6.055,148.858
C00638=1178.976,72.193,-49.558,-179.232,6.054,148.859
C00639=1178.982,71.944,-49.541,-179.235,6.052,148.859
C00640=1178.986,71.695,-49.524,-179.237,6.052,148.860
C00641=1178.991,71.446,-49.506,-179.240,6.051,148.860
C00642=1178.995,71.196,-49.490,-179.243,6.049,148.861
C00643=1179.001,70.947,-49.473,-179.245,6.049,148.862
C00644=1179.006,70.698,-49.456,-179.249,6.047,148.862
C00645=1179.010,70.448,-49.439,-179.251,6.047,148.863
C00646=1179.015,70.198,-49.422,-179.253,6.046,148.863
C00647=1179.021,69.949,-49.406,-179.256,6.044,148.864
C00648=1179.026,69.700,-49.388,-179.259,6.044,148.864
C00649=1179.030,69.450,-49.372,-179.261,6.043,148.865
C00650=1179.035,69.201,-49.355,-179.264,6.042,148.865
C00651=1179.041,68.952,-49.338,-179.266,6.041,148.866
C00652=1179.045,68.702,-49.322,-179.269,6.039,148.867
C00653=1179.049,68.453,-49.305,-179.272,6.038,148.867
C00654=1179.055,68.204,-49.288,-179.274,6.038,148.868
C00655=1179.060,67.954,-49.271,-179.277,6.036,148.868
C00656=1179.065,67.704,-49.254,-179.280,6.036,148.869
C00657=1179.070,67.455,-49.238,-179.282,6.035,148.869
C00658=1179.075,67.206,-49.221,-179.285,6.034,148.870
C00659=1179.080,66.956,-49.204,-179.287,6.033,148.870
C00660=1179.085,66.707,-49.188,-179.290,6.031,148.871
C00661=1179.089,66.458,-49.171,-179.292,6.030,148.871
C00662=1179.095,66.208,-49.154,-179.295,6.030,148.872
C00663=1179.100,65.959,-49.137,-179.298,6.028,148.872
C00664=1179.104,65.710,-49.121,-179.300,6.028,148.873
C00665=1179.109,65.460,-49.104,-179.303,6.027,148.874
C00666=1179.114,65.211,-49.087,-179.306,6.025,148.874
C00667=1179.119,64.961,-49.071,-179.308,6.025,148.875
C00668=1179.124,64.712,-49.054,-179.311,6.024,148.875
C00669=1179.130,64.463,-49.038,-179.314,6.023,148.876
C00670=1179.134,64.213,-49.021,-179.316,6.022,148.876
C00671=1179.138,63.964,-49.004,-179.319,6.021,148.877
C00672=1179.144,63.715,-48.988,-179.321,6.020,148.878
C00673=1179.149,63.465,-48.971,-179.324,6.019,148.878
C00674=1179.154,63.216,-48.955,-179.327,6.017,148.879
C00675=1179.159,62.966,-48.938,-179.329,6.017,148.879
C00676=1179.163,62.717,-48.922,-179.331,6.016,148.880
C00677=1179.168,62.468,-48.905,-179.335,6.015,148.880
C00678=1179.174,62.218,-48.889,-179.337,6.014,148.881
C00679=1179.179,61.969,-48.873,-179.339,6.013,148.881
C00680=1179.183,61.719,-48.856,-179.343,6.012,148.882
C00681=1179.188,61.470,-48.839,-179.345,6.011,148.883
C00682=1179.193,61.220,-48.824,-179.347,6.010,148.883
C00683=1179.198,60.971,-48.806,-179.350,6.009,148.884
C00684=1179.203,60.722,-48.790,-179.353,6.008,148.884
C00685=1179.208,60.472,-48.773,-179.355,6.007,148.885
C00686=1179.213,60.223,-48.758,-179.358,6.006,148.885
C00687=1179.218,59.973,-48.741,-179.360,6.005,148.886
C00688=1179.222,59.724,-48.724,-179.363,6.005,148.887
C00689=1179.228,59.474,-48.708,-179.366,6.004,148.887
C00690=1179.233,59.225,-48.692,-179.368,6.002,148.888
C00691=1179.238,58.976,-48.675,-179.371,6.002,148.888
C00692=1179.243,58.726,-48.659,-179.373,6.001,148.889
C00693=1179.248,58.477,-48.643,-179.376,6.000,148.889
C00694=1179.252,58.228,-48.626,-179.379,5.999,148.890
C00695=1179.258,57.978,-48.611,-179.381,5.998,148.891
C00696=1179.262,57.729,-48.594,-179.384,5.997,148.891
C00697=1179.268,57.479,-48.578,-179.387,5.996,148.892
C00698=1179.273,57.229,-48.561,-179.389,5.996,148.892
C00699=1179.278,56.981,-48.545,-179.392,5.994,148.893
C00700=1179.283,56.731,-48.529,-179.395,5.993,148.893
C00701=1179.288,56.482,-48.513,-179.397,5.993,148.894
C00702=1179.293,56.232,-48.497,-179.400,5.991,148.894
C00703=1179.298,55.983,-48.480,-179.402,5.990,148.895
C00704=1179.302,55.733,-48.464,-179.405,5.990,148.896
C00705=1179.307,55.484,-48.448,-179.407,5.989,148.896
C00706=1179.312,55.234,-48.432,-179.410,5.988,148.897
C00707=1179.317,54.985,-48.416,-179.413,5.987,148.897
C00708=1179.323,54.717,-48.399,-179.415,5.986,148.898
C00709=1179.328,54.447,-48.382,-179.418,5.985,148.898
C00710=1179.333,54.180,-48.364,-179.421,5.984,148.899
C00711=1179.339,53.911,-48.347,-179.424,5.983,148.900
C00712=1179.343,53.661,-48.331,-179.426,5.982,148.900
C00713=1179.349,53.412,-48.315,-179.429,5.982,148.901
C00714=1179.353,53.162,-48.299,-179.431,5.980,148.901
C00715=1179.358,52.913,-48.282,-179.434,5.979,148.902
C00716=1179.363,52.663,-48.266,-179.437,5.979,148.903
C00717=1179.368,52.415,-48.250,-179.439,5.977,148.903
C00718=1179.374,52.165,-48.234,-179.442,5.977,148.904
C00719=1179.378,51.915,-48.218,-179.444,5.976,148.904
C00720=1179.383,51.666,-48.202,-179.447,5.975,148.905
C00721=1179.388,51.416,-48.186,-179.450,5.974,148.906
C00722=1179.394,51.167,-48.171,-179.452,5.973,148.906
C00723=1179.399,50.918,-48.154,-179.455,5.973,148.907
C00724=1179.404,50.668,-48.138,-179.457,5.972,148.907
C00725=1179.409,50.419,-48.122,-179.460,5.970,148.908
C00726=1179.413,50.169,-48.106,-179.462,5.970,148.908
C00727=1179.419,49.920,-48.091,-179.465,5.969,148.909
C00728=1179.423,49.670,-48.076,-179.468,5.969,148.910
C00729=1179.428,49.421,-48.059,-179.470,5.967,148.910
C00730=1179.433,49.172,-48.043,-179.473,5.966,148.911
C00731=1179.438,48.921,-48.027,-179.475,5.965,148.911
C00732=1179.443,48.673,-48.011,-179.478,5.964,148.912
C00733=1179.449,48.423,-47.995,-179.481,5.964,148.912
C00734=1179.453,48.173,-47.979,-179.483,5.963,148.913
C00735=1179.458,47.924,-47.964,-179.486,5.962,148.914
C00736=1179.463,47.675,-47.948,-179.489,5.961,148.914
C00737=1179.468,47.425,-47.932,-179.491,5.960,148.915
C00738=1179.473,47.176,-47.917,-179.494,5.960,148.915
C00739=1179.479,46.926,-47.901,-179.496,5.959,148.916
C00740=1179.483,46.677,-47.884,-179.499,5.957,148.916
C00741=1179.488,46.428,-47.869,-179.501,5.956,148.917
C00742=1179.493,46.178,-47.854,-179.504,5.956,148.918
C00743=1179.498,45.928,-47.838,-179.507,5.955,148.918
C00744=1179.503,45.679,-47.822,-179.509,5.955,148.919
C00745=1179.509,45.429,-47.807,-179.512,5.953,148.919
C00746=1179.512,45.180,-47.791,-179.514,5.952,148.920
C00747=1179.518,44.931,-47.775,-179.517,5.952,148.920
C00748=1179.523,44.682,-47.759,-179.520,5.951,148.921
C00749=1179.528,44.431,-47.743,-179.522,5.950,148.922
C00750=1179.533,44.182,-47.728,-179.525,5.949,148.922
C00751=1179.538,43.933,-47.713,-179.527,5.948,148.923
C00752=1179.543,43.684,-47.697,-179.530,5.948,148.923
C00753=1179.548,43.433,-47.681,-179.533,5.947,148.924
C00754=1179.553,43.184,-47.666,-179.535,5.946,148.924
C00755=1179.558,42.936,-47.650,-179.538,5.945,148.925
C00756=1179.563,42.685,-47.634,-179.540,5.944,148.926
C00757=1179.568,42.436,-47.618,-179.542,5.944,148.926
C00758=1179.573,42.187,-47.604,-179.546,5.942,148.927
C00759=1179.578,41.938,-47.588,-179.548,5.942,148.927
C00760=1179.583,41.687,-47.572,-179.551,5.941,148.928
C00761=1179.588,41.438,-47.557,-179.553,5.940,148.928
C00762=1179.593,41.189,-47.541,-179.555,5.940,148.929
C00763=1179.598,40.940,-47.526,-179.559,5.938,148.930
C00764=1179.602,40.690,-47.510,-179.561,5.938,148.930
C00765=1179.608,40.440,-47.495,-179.563,5.937,148.931
C00766=1179.613,40.191,-47.479,-179.565,5.936,148.931
C00767=1179.618,39.942,-47.464,-179.569,5.935,148.932
C00768=1179.623,39.692,-47.449,-179.571,5.934,148.933
C00769=1179.628,39.442,-47.433,-179.574,5.933,148.933
C00770=1179.633,39.193,-47.418,-179.576,5.933,148.934
C00771=1179.638,38.943,-47.403,-179.579,5.932,148.935
C00772=1179.644,38.694,-47.387,-179.582,5.931,148.935
C00773=1179.648,38.445,-47.372,-179.584,5.930,148.936
C00774=1179.653,38.195,-47.356,-179.586,5.929,148.936
C00775=1179.658,37.946,-47.341,-179.589,5.929,148.937
C00776=1179.663,37.696,-47.326,-179.592,5.928,148.937
C00777=1179.669,37.447,-47.310,-179.594,5.928,148.938
C00778=1179.673,37.198,-47.295,-179.597,5.926,148.939
C00779=1179.678,36.948,-47.279,-179.600,5.926,148.939
C00780=1179.683,36.698,-47.265,-179.602,5.925,148.940
C00781=1179.688,36.448,-47.249,-179.604,5.924,148.940
C00782=1179.693,36.199,-47.234,-179.607,5.923,148.941
C00783=1179.698,35.950,-47.219,-179.610,5.922,148.941
C00784=1179.704,35.701,-47.203,-179.612,5.922,148.942
C00785=1179.709,35.451,-47.189,-179.615,5.921,148.943
C00786=1179.714,35.201,-47.173,-179.617,5.920,148.943
C00787=1179.718,34.952,-47.158,-179.620,5.920,148.944
C00788=1179.724,34.702,-47.142,-179.622,5.919,148.944
C00789=1179.728,34.453,-47.127,-179.625,5.918,148.945
C00790=1179.734,34.203,-47.113,-179.627,5.917,148.946
C00791=1179.739,33.954,-47.098,-179.630,5.916,148.946
C00792=1179.744,33.705,-47.082,-179.633,5.916,148.947
C00793=1179.748,33.455,-47.067,-179.635,5.915,148.947
C00794=1179.754,33.205,-47.052,-179.638,5.914,148.948
C00795=1179.758,32.956,-47.037,-179.641,5.913,148.949
C00796=1179.764,32.706,-47.021,-179.643,5.912,148.949
C00797=1179.769,32.457,-47.007,-179.646,5.912,148.950
C00798=1179.773,32.208,-46.992,-179.648,5.911,148.950
C00799=1179.779,31.958,-46.976,-179.650,5.910,148.951
C00800=1179.784,31.708,-46.962,-179.653,5.910,148.952
C00801=1179.789,31.459,-46.946,-179.656,5.908,148.952
C00802=1179.794,31.210,-46.931,-179.658,5.908,148.953
C00803=1179.799,30.959,-46.916,-179.661,5.907,148.953
C00804=1179.803,30.710,-46.901,-179.663,5.906,148.954
C00805=1179.809,30.461,-46.886,-179.666,5.906,148.955
C00806=1179.814,30.211,-46.871,-179.669,5.905,148.955
C00807=1179.818,29.962,-46.856,-179.671,5.905,148.956
C00808=1179.824,29.712,-46.841,-179.674,5.903,148.956
C00809=1179.829,29.463,-46.826,-179.677,5.903,148.957
C00810=1179.833,29.214,-46.811,-179.679,5.902,148.957
C00811=1179.839,28.964,-46.797,-179.681,5.901,148.958
C00812=1179.844,28.695,-46.781,-179.684,5.901,148.959
C00813=1179.850,28.426,-46.764,-179.687,5.900,148.959
C00814=1179.855,28.158,-46.748,-179.689,5.899,148.960
C00815=1179.861,27.888,-46.732,-179.692,5.898,148.961
C00816=1179.866,27.639,-46.718,-179.695,5.898,148.961
C00817=1179.870,27.390,-46.703,-179.697,5.896,148.962
C00818=1179.876,27.140,-46.688,-179.700,5.896,148.962
C00819=1179.881,26.891,-46.673,-179.703,5.895,148.963
C00820=1179.886,26.641,-46.658,-179.705,5.894,148.964
C00821=1179.891,26.391,-46.643,-179.708,5.894,148.964
C00822=1179.896,26.142,-46.629,-179.710,5.893,148.965
C00823=1179.901,25.893,-46.614,-179.712,5.892,148.965
C00824=1179.906,25.643,-46.599,-179.715,5.892,148.966
C00825=1179.911,25.394,-46.584,-179.718,5.891,148.967
C00826=1179.916,25.144,-46.569,-179.720,5.890,148.967
C00827=1179.921,24.895,-46.554,-179.723,5.889,148.968
C00828=1179.926,24.645,-46.540,-179.726,5.889,148.969
C00829=1179.931,24.395,-46.525,-179.728,5.888,148.969
C00830=1179.936,24.146,-46.510,-179.731,5.887,148.970
C00831=1179.941,23.896,-46.496,-179.733,5.887,148.970
C00832=1179.946,23.647,-46.480,-179.735,5.886,148.971
C00833=1179.951,23.397,-46.466,-179.738,5.886,148.971
C00834=1179.956,23.147,-46.452,-179.741,5.884,148.972
C00835=1179.961,22.898,-46.437,-179.743,5.883,148.973
C00836=1179.967,22.648,-46.422,-179.746,5.883,148.973
C00837=1179.972,22.399,-46.408,-179.749,5.882,148.974
C00838=1179.977,22.150,-46.393,-179.751,5.882,148.974
C00839=1179.982,21.900,-46.379,-179.753,5.881,148.975
C00840=1179.987,21.651,-46.365,-179.756,5.881,148.976
C00841=1179.992,21.401,-46.349,-179.758,5.880,148.976
C00842=1179.997,21.152,-46.335,-179.761,5.879,148.977
C00843=1180.002,20.902,-46.320,-179.763,5.878,148.977
C00844=1180.007,20.653,-46.305,-179.766,5.877,148.978
C00845=1180.012,20.403,-46.291,-179.769,5.877,148.979
C00846=1180.016,20.153,-46.277,-179.771,5.876,148.979
C00847=1180.022,19.904,-46.261,-179.774,5.875,148.980
C00848=1180.027,19.654,-46.247,-179.776,5.875,148.981
C00849=1180.032,19.405,-46.233,-179.779,5.874,148.981
C00850=1180.037,19.156,-46.219,-179.781,5.873,148.982
C00851=1180.042,18.906,-46.205,-179.784,5.873,148.982
C00852=1180.047,18.657,-46.190,-179.786,5.872,148.983
C00853=1180.052,18.407,-46.175,-179.789,5.872,148.984
C00854=1180.058,18.157,-46.160,-179.791,5.871,148.984
C00855=1180.063,17.907,-46.146,-179.794,5.869,148.985
C00856=1180.068,17.658,-46.132,-179.797,5.869,148.985
C00857=1180.073,17.409,-46.117,-179.799,5.869,148.986
C00858=1180.078,17.160,-46.103,-179.802,5.868,148.986
C00859=1180.083,16.910,-46.089,-179.804,5.867,148.987
C00860=1180.088,16.660,-46.074,-179.807,5.867,148.988
C00861=1180.093,16.410,-46.060,-179.809,5.866,148.988
C00862=1180.098,16.161,-46.046,-179.812,5.865,148.989
C00863=1180.102,15.912,-46.031,-179.814,5.865,148.990
C00864=1180.108,15.663,-46.017,-179.816,5.864,148.990
C00865=1180.113,15.413,-46.003,-179.819,5.864,148.991
C00866=1180.118,15.163,-45.988,-179.822,5.863,148.991
C00867=1180.123,14.913,-45.973,-179.824,5.862,148.992
C00868=1180.128,14.663,-45.959,-179.827,5.862,148.993
C00869=1180.134,14.414,-45.945,-179.829,5.861,148.993
C00870=1180.139,14.165,-45.931,-179.832,5.860,148.994
C00871=1180.144,13.915,-45.917,-179.835,5.859,148.994
C00872=1180.149,13.665,-45.902,-179.837,5.859,148.995
C00873=1180.154,13.416,-45.888,-179.840,5.858,148.996
C00874=1180.159,13.167,-45.874,-179.842,5.857,148.996
C00875=1180.164,12.917,-45.860,-179.845,5.857,148.997
C00876=1180.169,12.667,-45.846,-179.847,5.856,148.998
C00877=1180.174,12.417,-45.831,-179.850,5.855,148.998
C00878=1180.179,12.168,-45.817,-179.852,5.855,148.999
C00879=1180.185,11.919,-45.803,-179.855,5.855,148.999
C00880=1180.190,11.669,-45.789,-179.857,5.854,149.000
C00881=1180.194,11.420,-45.775,-179.860,5.853,149.001
C00882=1180.199,11.170,-45.761,-179.862,5.853,149.001
C00883=1180.204,10.921,-45.747,-179.865,5.852,149.002
C00884=1180.209,10.671,-45.733,-179.867,5.851,149.002
C00885=1180.214,10.421,-45.719,-179.870,5.851,149.003
C00886=1180.219,10.172,-45.704,-179.872,5.850,149.004
C00887=1180.225,9.923,-45.690,-179.875,5.850,149.004
C00888=1180.230,9.673,-45.676,-179.877,5.849,149.005
C00889=1180.235,9.423,-45.662,-179.879,5.848,149.005
C00890=1180.240,9.174,-45.648,-179.882,5.848,149.006
C00891=1180.245,8.925,-45.634,-179.885,5.847,149.007
C00892=1180.250,8.675,-45.619,-179.887,5.846,149.007
C00893=1180.255,8.425,-45.606,-179.890,5.845,149.008
C00894=1180.260,8.176,-45.592,-179.893,5.845,149.009
C00895=1180.265,7.926,-45.578,-179.895,5.844,149.009
C00896=1180.270,7.676,-45.564,-179.898,5.843,149.010
C00897=1180.275,7.427,-45.550,-179.900,5.843,149.010
C00898=1180.281,7.178,-45.536,-179.902,5.842,149.011
C00899=1180.286,6.927,-45.522,-179.905,5.842,149.012
C00900=1180.290,6.678,-45.508,-179.908,5.841,149.012
C00901=1180.296,6.429,-45.495,-179.910,5.840,149.013
C00902=1180.301,6.179,-45.480,-179.913,5.840,149.013
C00903=1180.306,5.930,-45.466,-179.915,5.839,149.014
C00904=1180.311,5.680,-45.453,-179.918,5.839,149.015
C00905=1180.316,5.430,-45.439,-179.920,5.838,149.015
C00906=1180.321,5.181,-45.425,-179.923,5.837,149.016
C00907=1180.326,4.932,-45.411,-179.925,5.837,149.017
C00908=1180.331,4.682,-45.397,-179.928,5.836,149.017
C00909=1180.336,4.432,-45.383,-179.930,5.836,149.018
C00910=1180.342,4.183,-45.369,-179.933,5.835,149.018
C00911=1180.346,3.933,-45.356,-179.935,5.834,149.019
C00912=1180.351,3.683,-45.342,-179.938,5.834,149.020
C00913=1180.357,3.434,-45.328,-179.940,5.833,149.020
C00914=1180.362,3.184,-45.314,-179.942,5.833,149.021
C00915=1180.366,2.935,-45.300,-179.945,5.832,149.021
C00916=1180.372,2.666,-45.285,-179.948,5.832,149.022
C00917=1180.378,2.397,-45.270,-179.950,5.831,149.023
C00918=1180.383,2.127,-45.255,-179.953,5.831,149.023
C00919=1180.388,1.858,-45.240,-179.956,5.830,149.024
C00920=1180.394,1.608,-45.227,-179.958,5.829,149.025
C00921=1180.398,1.359,-45.214,-179.961,5.829,149.025
C00922=1180.404,1.109,-45.200,-179.963,5.828,149.026
C00923=1180.409,0.860,-45.186,-179.965,5.828,149.026
C00924=1180.414,0.610,-45.172,-179.968,5.827,149.027
C00925=1180.419,0.361,-45.159,-179.971,5.827,149.028
C00926=1180.424,0.111,-45.145,-179.973,5.826,149.029
C00927=1180.430,-0.139,-45.132,-179.976,5.825,149.029
C00928=1180.434,-0.388,-45.118,-179.978,5.825,149.030
C00929=1180.439,-0.638,-45.104,-179.981,5.824,149.030
C00930=1180.445,-0.888,-45.091,-179.983,5.824,149.031
C00931=1180.449,-1.137,-45.077,-179.986,5.823,149.032
C00932=1180.455,-1.387,-45.064,-179.988,5.823,149.032
C00933=1180.460,-1.636,-45.049,-179.990,5.822,149.033
C00934=1180.465,-1.886,-45.037,-179.993,5.821,149.033
C00935=1180.470,-2.135,-45.023,-179.996,5.821,149.034
C00936=1180.476,-2.386,-45.009,-179.998,5.820,149.035
C00937=1180.480,-2.634,-44.996,179.999,5.820,149.035
C00938=1180.486,-2.885,-44.982,179.997,5.819,149.036
C00939=1180.491,-3.133,-44.969,179.995,5.818,149.036
C00940=1180.496,-3.384,-44.955,179.992,5.818,149.037
C00941=1180.501,-3.633,-44.941,179.989,5.817,149.038
C00942=1180.506,-3.883,-44.928,179.987,5.817,149.038
C00943=1180.511,-4.132,-44.914,179.984,5.816,149.039
C00944=1180.516,-4.382,-44.902,179.982,5.815,149.040
C00945=1180.521,-4.631,-44.888,179.979,5.815,149.040
C00946=1180.526,-4.881,-44.875,179.977,5.814,149.041
C00947=1180.532,-5.130,-44.861,179.974,5.814,149.041
C00948=1180.537,-5.380,-44.847,179.972,5.813,149.042
C00949=1180.542,-5.629,-44.835,179.969,5.812,149.043
C00950=1180.547,-5.879,-44.820,179.967,5.812,149.043
C00951=1180.552,-6.128,-44.808,179.964,5.811,149.044
C00952=1180.557,-6.378,-44.793,179.962,5.812,149.045
C00953=1180.562,-6.627,-44.781,179.960,5.811,149.045
C00954=1180.567,-6.878,-44.767,179.957,5.811,149.046
C00955=1180.572,-7.126,-44.754,179.955,5.810,149.046
C00956=1180.577,-7.377,-44.740,179.952,5.809,149.047
C00957=1180.583,-7.626,-44.728,179.950,5.809,149.048
C00958=1180.588,-7.876,-44.714,179.947,5.808,149.048
C00959=1180.593,-8.125,-44.701,179.945,5.807,149.049
C00960=1180.598,-8.375,-44.687,179.942,5.807,149.049
C00961=1180.603,-8.624,-44.674,179.940,5.807,149.050
C00962=1180.608,-8.875,-44.660,179.937,5.806,149.051
C00963=1180.613,-9.124,-44.648,179.935,5.805,149.051
C00964=1180.619,-9.373,-44.634,179.932,5.805,149.052
C00965=1180.623,-9.623,-44.621,179.929,5.804,149.053
C00966=1180.629,-9.872,-44.608,179.927,5.803,149.053
C00967=1180.634,-10.123,-44.595,179.925,5.803,149.054
C00968=1180.639,-10.372,-44.581,179.923,5.803,149.055
C00969=1180.644,-10.622,-44.568,179.920,5.803,149.055
C00970=1180.649,-10.871,-44.555,179.918,5.802,149.056
C00971=1180.655,-11.120,-44.542,179.915,5.802,149.056
C00972=1180.659,-11.370,-44.528,179.913,5.801,149.057
C00973=1180.665,-11.620,-44.515,179.910,5.800,149.058
C00974=1180.669,-11.870,-44.502,179.908,5.800,149.058
C00975=1180.675,-12.119,-44.489,179.905,5.799,149.059
C00976=1180.680,-12.369,-44.476,179.903,5.799,149.059
C00977=1180.684,-12.618,-44.463,179.900,5.798,149.060
C00978=1180.690,-12.867,-44.450,179.897,5.798,149.061
C00979=1180.695,-13.118,-44.437,179.895,5.797,149.061
C00980=1180.700,-13.367,-44.424,179.893,5.796,149.062
C00981=1180.706,-13.616,-44.411,179.891,5.797,149.063
C00982=1180.710,-13.866,-44.398,179.888,5.796,149.063
C00983=1180.716,-14.115,-44.384,179.886,5.795,149.064
C00984=1180.720,-14.366,-44.371,179.883,5.795,149.065
C00985=1180.726,-14.615,-44.358,179.880,5.794,149.065
C00986=1180.731,-14.864,-44.345,179.878,5.794,149.066
C00987=1180.736,-15.114,-44.332,179.876,5.793,149.066
C00988=1180.741,-15.364,-44.320,179.873,5.793,149.067
C00989=1180.747,-15.613,-44.306,179.871,5.792,149.068
C00990=1180.751,-15.863,-44.293,179.868,5.791,149.068
C00991=1180.757,-16.113,-44.281,179.865,5.791,149.069
C00992=1180.762,-16.362,-44.268,179.864,5.791,149.069
C00993=1180.767,-16.612,-44.255,179.861,5.790,149.070
C00994=1180.772,-16.862,-44.242,179.859,5.790,149.071
C00995=1180.777,-17.110,-44.229,179.856,5.790,149.071
C00996=1180.782,-17.361,-44.215,179.854,5.789,149.072
C00997=1180.787,-17.610,-44.203,179.851,5.788,149.073
C00998=1180.792,-17.859,-44.190,179.848,5.788,149.073
C00999=1180.798,-18.110,-44.176,179.846,5.787,149.074
C01000=1180.803,-18.359,-44.164,179.844,5.787,149.074
C01001=1180.808,-18.608,-44.151,179.841,5.786,149.075
C01002=1180.812,-18.858,-44.138,179.839,5.786,149.076
C01003=1180.818,-19.108,-44.125,179.837,5.786,149.076
C01004=1180.823,-19.357,-44.113,179.834,5.785,149.077
C01005=1180.829,-19.607,-44.100,179.831,5.785,149.078
C01006=1180.833,-19.857,-44.088,179.829,5.784,149.078
C01007=1180.839,-20.107,-44.074,179.826,5.783,149.079
C01008=1180.844,-20.356,-44.062,179.824,5.783,149.080
C01009=1180.849,-20.606,-44.049,179.822,5.782,149.080
C01010=1180.854,-20.856,-44.036,179.820,5.782,149.081
C01011=1180.860,-21.105,-44.023,179.817,5.782,149.081
C01012=1180.865,-21.355,-44.011,179.815,5.781,149.082
C01013=1180.869,-21.605,-43.998,179.812,5.781,149.083
C01014=1180.875,-21.854,-43.985,179.809,5.780,149.083
C01015=1180.880,-22.103,-43.972,179.807,5.780,149.084
C01016=1180.885,-22.352,-43.960,179.805,5.779,149.084
C01017=1180.891,-22.603,-43.947,179.802,5.779,149.085
C01018=1180.896,-22.853,-43.934,179.800,5.779,149.086
C01019=1180.901,-23.102,-43.922,179.798,5.778,149.086
C01020=1180.906,-23.372,-43.908,179.795,5.778,149.087
C01021=1180.912,-23.641,-43.894,179.792,5.777,149.088
C01022=1180.917,-23.911,-43.880,179.790,5.777,149.088
C01023=1180.923,-24.182,-43.867,179.787,5.776,149.089
C01024=1180.928,-24.431,-43.854,179.784,5.776,149.090
C01025=1180.933,-24.680,-43.842,179.782,5.775,149.090
C01026=1180.938,-24.929,-43.829,179.780,5.775,149.091
C01027=1180.944,-25.179,-43.816,179.777,5.774,149.092
C01028=1180.948,-25.429,-43.804,179.774,5.774,149.092
C01029=1180.954,-25.679,-43.792,179.772,5.773,149.093
C01030=1180.959,-25.928,-43.779,179.770,5.773,149.094
C01031=1180.964,-26.177,-43.766,179.767,5.773,149.094
C01032=1180.970,-26.428,-43.754,179.765,5.772,149.095
C01033=1180.974,-26.678,-43.741,179.762,5.771,149.095
C01034=1180.980,-26.927,-43.728,179.760,5.771,149.096
C01035=1180.985,-27.176,-43.716,179.758,5.770,149.097
C01036=1180.990,-27.426,-43.704,179.756,5.771,149.097
C01037=1180.995,-27.676,-43.691,179.753,5.770,149.098
C01038=1181.000,-27.926,-43.678,179.750,5.770,149.099
C01039=1181.005,-28.175,-43.666,179.748,5.769,149.099
C01040=1181.010,-28.425,-43.654,179.745,5.768,149.100
C01041=1181.015,-28.674,-43.641,179.743,5.768,149.101
C01042=1181.021,-28.924,-43.629,179.741,5.767,149.101
C01043=1181.026,-29.173,-43.617,179.738,5.767,149.102
C01044=1181.031,-29.423,-43.604,179.736,5.767,149.102
C01045=1181.036,-29.673,-43.592,179.734,5.766,149.103
C01046=1181.041,-29.923,-43.579,179.731,5.766,149.104
C01047=1181.046,-30.172,-43.567,179.728,5.765,149.104
C01048=1181.052,-30.422,-43.555,179.726,5.764,149.105
C01049=1181.057,-30.671,-43.542,179.724,5.765,149.105
C01050=1181.062,-30.921,-43.530,179.721,5.764,149.106
C01051=1181.067,-31.170,-43.518,179.719,5.764,149.107
C01052=1181.072,-31.420,-43.505,179.717,5.763,149.107
C01053=1181.077,-31.670,-43.493,179.714,5.763,149.108
C01054=1181.082,-31.920,-43.480,179.711,5.762,149.109
C01055=1181.088,-32.170,-43.468,179.710,5.762,149.109
C01056=1181.093,-32.419,-43.456,179.707,5.762,149.110
C01057=1181.098,-32.668,-43.443,179.704,5.761,149.111
C01058=1181.103,-32.918,-43.431,179.702,5.760,149.111
C01059=1181.109,-33.168,-43.419,179.699,5.760,149.112
C01060=1181.114,-33.418,-43.407,179.697,5.760,149.112
C01061=1181.119,-33.667,-43.394,179.695,5.760,149.113
C01062=1181.125,-33.917,-43.382,179.693,5.759,149.114
C01063=1181.129,-34.166,-43.370,179.690,5.759,149.114
C01064=1181.134,-34.416,-43.358,179.687,5.758,149.115
C01065=1181.139,-34.666,-43.345,179.685,5.757,149.115
C01066=1181.144,-34.916,-43.334,179.683,5.758,149.116
C01067=1181.149,-35.165,-43.321,179.680,5.757,149.117
C01068=1181.155,-35.415,-43.309,179.678,5.756,149.117
C01069=1181.160,-35.664,-43.296,179.675,5.756,149.118
C01070=1181.165,-35.914,-43.285,179.673,5.756,149.119
C01071=1181.171,-36.163,-43.272,179.671,5.756,149.119
C01072=1181.175,-36.413,-43.261,179.669,5.755,149.120
C01073=1181.181,-36.663,-43.249,179.666,5.755,149.121
C01074=1181.186,-36.912,-43.236,179.663,5.754,149.121
C01075=1181.191,-37.162,-43.224,179.661,5.753,149.122
C01076=1181.196,-37.412,-43.212,179.659,5.754,149.122
C01077=1181.202,-37.662,-43.200,179.656,5.753,149.123
C01078=1181.207,-37.911,-43.188,179.654,5.753,149.124
C01079=1181.212,-38.160,-43.176,179.651,5.752,149.124
C01080=1181.217,-38.410,-43.164,179.649,5.752,149.125
C01081=1181.222,-38.660,-43.151,179.647,5.752,149.125
C01082=1181.228,-38.910,-43.140,179.645,5.751,149.126
C01083=1181.233,-39.160,-43.128,179.642,5.751,149.127
C01084=1181.238,-39.409,-43.115,179.639,5.750,149.128
C01085=1181.243,-39.659,-43.104,179.637,5.750,149.128
C01086=1181.248,-39.909,-43.092,179.635,5.750,149.129
C01087=1181.253,-40.158,-43.079,179.632,5.749,149.129
C01088=1181.259,-40.408,-43.067,179.630,5.749,149.130
C01089=1181.264,-40.657,-43.056,179.627,5.748,149.131
C01090=1181.269,-40.907,-43.044,179.625,5.748,149.131
C01091=1181.274,-41.157,-43.032,179.623,5.748,149.132
C01092=1181.280,-41.407,-43.020,179.621,5.747,149.133
C01093=1181.284,-41.656,-43.008,179.618,5.747,149.133
C01094=1181.289,-41.906,-42.996,179.616,5.746,149.134
C01095=1181.295,-42.155,-42.984,179.614,5.746,149.134
C01096=1181.300,-42.405,-42.972,179.611,5.746,149.135
C01097=1181.305,-42.655,-42.961,179.609,5.745,149.136
C01098=1181.310,-42.904,-42.948,179.606,5.745,149.136
C01099=1181.315,-43.154,-42.936,179.603,5.744,149.137
C01100=1181.321,-43.404,-42.924,179.601,5.745,149.138
C01101=1181.326,-43.653,-42.914,179.599,5.744,149.138
C01102=1181.331,-43.902,-42.901,179.597,5.743,149.139
C01103=1181.337,-44.152,-42.889,179.594,5.743,149.140
C01104=1181.341,-44.402,-42.878,179.592,5.743,149.140
C01105=1181.347,-44.652,-42.866,179.590,5.743,149.141
C01106=1181.352,-44.902,-42.854,179.587,5.742,149.141
C01107=1181.357,-45.151,-42.842,179.585,5.741,149.142
C01108=1181.362,-45.401,-42.830,179.583,5.742,149.143
C01109=1181.368,-45.651,-42.818,179.580,5.741,149.143
C01110=1181.372,-45.900,-42.807,179.578,5.740,149.144
C01111=1181.378,-46.150,-42.795,179.575,5.740,149.144
C01112=1181.383,-46.400,-42.783,179.573,5.740,149.145
C01113=1181.388,-46.649,-42.772,179.571,5.739,149.146
C01114=1181.393,-46.899,-42.760,179.568,5.739,149.146
C01115=1181.399,-47.148,-42.748,179.566,5.739,149.147
C01116=1181.404,-47.398,-42.736,179.563,5.738,149.148
C01117=1181.409,-47.648,-42.725,179.561,5.738,149.148
C01118=1181.414,-47.898,-42.713,179.559,5.738,149.149
C01119=1181.419,-48.148,-42.701,179.556,5.737,149.150
C01120=1181.425,-48.398,-42.690,179.554,5.737,149.150
C01121=1181.430,-48.646,-42.679,179.552,5.737,149.151
C01122=1181.435,-48.896,-42.667,179.549,5.736,149.152
C01123=1181.441,-49.146,-42.655,179.547,5.736,149.152
C01124=1181.446,-49.417,-42.642,179.544,5.735,149.153
C01125=1181.452,-49.686,-42.629,179.542,5.735,149.153
C01126=1181.458,-49.957,-42.617,179.539,5.734,149.154
C01127=1181.463,-50.228,-42.604,179.537,5.735,149.155
C01128=1181.468,-50.477,-42.593,179.534,5.734,149.156
C01129=1181.474,-50.727,-42.581,179.532,5.733,149.156
C01130=1181.478,-50.976,-42.570,179.529,5.733,149.157
C01131=1181.484,-51.226,-42.558,179.527,5.733,149.157
C01132=1181.488,-51.476,-42.547,179.525,5.733,149.158
C01133=1181.494,-51.726,-42.535,179.522,5.732,149.159
C01134=1181.499,-51.975,-42.524,179.520,5.732,149.159
C01135=1181.505,-52.224,-42.512,179.518,5.732,149.160
C01136=1181.509,-52.474,-42.501,179.515,5.731,149.160
C01137=1181.515,-52.724,-42.489,179.513,5.731,149.161
C01138=1181.519,-52.974,-42.478,179.511,5.730,149.162
C01139=1181.525,-53.223,-42.466,179.509,5.730,149.162
C01140=1181.530,-53.473,-42.455,179.506,5.730,149.163
C01141=1181.536,-53.723,-42.444,179.504,5.729,149.164
C01142=1181.541,-53.973,-42.432,179.502,5.730,149.164
C01143=1181.546,-54.223,-42.420,179.499,5.729,149.165
C01144=1181.551,-54.472,-42.410,179.497,5.728,149.165
C01145=1181.557,-54.722,-42.398,179.494,5.728,149.166
C01146=1181.561,-54.971,-42.386,179.492,5.728,149.167
C01147=1181.567,-55.221,-42.374,179.490,5.727,149.167
C01148=1181.572,-55.471,-42.363,179.487,5.727,149.168
C01149=1181.578,-55.720,-42.352,179.484,5.727,149.169
C01150=1181.583,-55.970,-42.341,179.483,5.727,149.169
C01151=1181.587,-56.220,-42.330,179.480,5.726,149.170
C01152=1181.593,-56.470,-42.318,179.478,5.726,149.171
C01153=1181.598,-56.719,-42.307,179.476,5.726,149.171
C01154=1181.603,-56.969,-42.295,179.473,5.725,149.172
C01155=1181.608,-57.218,-42.284,179.471,5.725,149.172
C01156=1181.614,-57.469,-42.273,179.468,5.724,149.173
C01157=1181.619,-57.718,-42.262,179.466,5.724,149.174
C01158=1181.624,-57.967,-42.250,179.464,5.724,149.174
C01159=1181.629,-58.217,-42.239,179.462,5.723,149.175
C01160=1181.634,-58.467,-42.227,179.459,5.724,149.176
C01161=1181.640,-58.717,-42.216,179.457,5.723,149.176
C01162=1181.645,-58.966,-42.205,179.455,5.722,149.177
C01163=1181.650,-59.216,-42.194,179.452,5.722,149.177
C01164=1181.656,-59.465,-42.182,179.450,5.722,149.178
C01165=1181.661,-59.715,-42.172,179.448,5.722,149.179
C01166=1181.665,-59.965,-42.160,179.445,5.721,149.179
C01167=1181.671,-60.215,-42.149,179.443,5.721,149.180
C01168=1181.676,-60.464,-42.138,179.441,5.721,149.180
C01169=1181.681,-60.714,-42.127,179.438,5.720,149.181
C01170=1181.686,-60.964,-42.115,179.436,5.721,149.182
C01171=1181.692,-61.213,-42.104,179.434,5.720,149.182
C01172=1181.697,-61.463,-42.094,179.431,5.719,149.183
C01173=1181.702,-61.713,-42.082,179.428,5.719,149.184
C01174=1181.708,-61.962,-42.071,179.427,5.719,149.184
C01175=1181.713,-62.212,-42.060,179.424,5.719,149.185
C01176=1181.718,-62.462,-42.048,179.422,5.718,149.186
C01177=1181.723,-62.711,-42.038,179.420,5.718,149.186
C01178=1181.728,-62.962,-42.027,179.417,5.718,149.187
C01179=1181.734,-63.211,-42.015,179.415,5.717,149.188
C01180=1181.739,-63.460,-42.004,179.413,5.717,149.188
C01181=1181.744,-63.711,-41.994,179.410,5.717,149.189
C01182=1181.749,-63.960,-41.982,179.408,5.716,149.189
C01183=1181.755,-64.209,-41.971,179.406,5.716,149.190
C01184=1181.760,-64.460,-41.960,179.403,5.716,149.191
C01185=1181.764,-64.709,-41.949,179.401,5.716,149.191
C01186=1181.770,-64.959,-41.939,179.399,5.715,149.192
C01187=1181.775,-65.209,-41.927,179.396,5.715,149.193
C01188=1181.780,-65.458,-41.915,179.394,5.715,149.193
C01189=1181.786,-65.708,-41.905,179.392,5.714,149.194
C01190=1181.790,-65.958,-41.894,179.390,5.714,149.194
C01191=1181.797,-66.207,-41.883,179.387,5.714,149.195
C01192=1181.801,-66.457,-41.872,179.385,5.713,149.196
C01193=1181.806,-66.707,-41.861,179.383,5.713,149.196
C01194=1181.812,-66.956,-41.850,179.380,5.713,149.197
C01195=1181.817,-67.207,-41.839,179.378,5.712,149.198
C01196=1181.823,-67.456,-41.828,179.376,5.713,149.198
C01197=1181.828,-67.706,-41.818,179.373,5.712,149.199
C01198=1181.832,-67.956,-41.806,179.371,5.711,149.199
C01199=1181.838,-68.205,-41.796,179.369,5.712,149.200
C01200=1181.843,-68.455,-41.784,179.367,5.711,149.201
C01201=1181.849,-68.705,-41.774,179.364,5.711,149.201
C01202=1181.854,-68.954,-41.763,179.362,5.711,149.202
C01203=1181.859,-69.204,-41.753,179.360,5.710,149.202
C01204=1181.864,-69.453,-41.741,179.357,5.710,149.203
C01205=1181.870,-69.704,-41.730,179.355,5.710,149.204
C01206=1181.875,-69.953,-41.719,179.353,5.709,149.204
C01207=1181.880,-70.203,-41.709,179.350,5.709,149.205
C01208=1181.885,-70.452,-41.698,179.348,5.709,149.206
C01209=1181.890,-70.702,-41.687,179.346,5.709,149.206
C01210=1181.896,-70.952,-41.677,179.343,5.708,149.207
C01211=1181.901,-71.202,-41.666,179.341,5.708,149.207
C01212=1181.907,-71.451,-41.655,179.339,5.708,149.208
C01213=1181.912,-71.701,-41.644,179.336,5.707,149.209
C01214=1181.917,-71.951,-41.633,179.335,5.707,149.209
C01215=1181.922,-72.201,-41.623,179.332,5.707,149.210
C01216=1181.927,-72.450,-41.612,179.329,5.706,149.211
C01217=1181.933,-72.700,-41.601,179.328,5.706,149.211
C01218=1181.937,-72.950,-41.590,179.325,5.706,149.212
C01219=1181.943,-73.199,-41.580,179.323,5.705,149.212
C01220=1181.948,-73.449,-41.569,179.321,5.706,149.213
C01221=1181.954,-73.699,-41.558,179.318,5.705,149.214
C01222=1181.959,-73.949,-41.547,179.316,5.705,149.214
C01223=1181.964,-74.198,-41.537,179.314,5.705,149.215
C01224=1181.969,-74.448,-41.526,179.311,5.704,149.216
C01225=1181.975,-74.698,-41.515,179.309,5.704,149.216
C01226=1181.980,-74.948,-41.505,179.307,5.704,149.217
C01227=1181.985,-75.197,-41.494,179.304,5.704,149.218
C01228=1181.991,-75.468,-41.482,179.303,5.704,149.218
C01229=1181.997,-75.739,-41.472,179.300,5.703,149.219
C01230=1182.002,-76.010,-41.460,179.297,5.703,149.220
C01231=1182.008,-76.281,-41.449,179.294,5.702,149.220
C01232=1182.013,-76.530,-41.438,179.292,5.703,149.221
C01233=1182.019,-76.781,-41.427,179.290,5.702,149.221
C01234=1182.024,-77.030,-41.416,179.288,5.701,149.222
C01235=1182.029,-77.280,-41.406,179.286,5.701,149.223
C01236=1182.034,-77.529,-41.395,179.283,5.701,149.223
C01237=1182.039,-77.780,-41.384,179.281,5.701,149.224
C01238=1182.045,-78.029,-41.374,179.279,5.701,149.225
C01239=1182.051,-78.279,-41.364,179.276,5.700,149.225
C01240=1182.056,-78.529,-41.353,179.274,5.700,149.226
C01241=1182.061,-78.778,-41.342,179.272,5.700,149.226
C01242=1182.066,-79.028,-41.332,179.269,5.699,149.227
C01243=1182.072,-79.278,-41.322,179.268,5.699,149.228
C01244=1182.076,-79.528,-41.312,179.265,5.699,149.228
C01245=1182.081,-79.777,-41.301,179.262,5.699,149.229
C01246=1182.087,-80.026,-41.290,179.261,5.699,149.230
C01247=1182.092,-80.276,-41.280,179.258,5.698,149.230
C01248=1182.097,-80.526,-41.270,179.256,5.697,149.231
C01249=1182.102,-80.776,-41.259,179.254,5.698,149.231
C01250=1182.108,-81.026,-41.249,179.251,5.697,149.232
C01251=1182.113,-81.276,-41.238,179.250,5.697,149.233
C01252=1182.118,-81.525,-41.228,179.247,5.697,149.233
C01253=1182.124,-81.774,-41.217,179.244,5.697,149.234
C01254=1182.129,-82.025,-41.207,179.243,5.697,149.234
C01255=1182.134,-82.274,-41.196,179.240,5.696,149.235
C01256=1182.139,-82.524,-41.186,179.238,5.695,149.236
C01257=1182.145,-82.774,-41.176,179.236,5.696,149.236
C01258=1182.150,-83.023,-41.166,179.233,5.695,149.237
C01259=1182.155,-83.273,-41.155,179.232,5.695,149.238
C01260=1182.160,-83.523,-41.145,179.229,5.695,149.238
C01261=1182.166,-83.773,-41.135,179.227,5.694,149.239
C01262=1182.171,-84.023,-41.124,179.225,5.695,149.239
C01263=1182.177,-84.272,-41.114,179.222,5.694,149.240
C01264=1182.182,-84.523,-41.104,179.220,5.694,149.241
C01265=1182.187,-84.772,-41.093,179.218,5.694,149.241
C01266=1182.192,-85.021,-41.084,179.215,5.693,149.242
C01267=1182.197,-85.272,-41.073,179.213,5.693,149.243
C01268=1182.203,-85.521,-41.063,179.211,5.693,149.243
C01269=1182.208,-85.771,-41.053,179.209,5.693,149.244
C01270=1182.213,-86.021,-41.042,179.206,5.693,149.244
C01271=1182.219,-86.270,-41.032,179.204,5.692,149.245
C01272=1182.224,-86.520,-41.022,179.202,5.692,149.246
C01273=1182.229,-86.770,-41.012,179.199,5.692,149.246
C01274=1182.234,-87.019,-41.002,179.198,5.692,149.247
C01275=1182.240,-87.269,-40.991,179.195,5.691,149.248
C01276=1182.245,-87.519,-40.981,179.193,5.691,149.248
C01277=1182.250,-87.768,-40.971,179.191,5.691,149.249
C01278=1182.255,-88.018,-40.961,179.188,5.691,149.249
C01279=1182.260,-88.268,-40.950,179.187,5.691,149.250
C01280=1182.266,-88.518,-40.940,179.184,5.690,149.251
C01281=1182.271,-88.767,-40.931,179.182,5.689,149.251
C01282=1182.276,-89.017,-40.920,179.180,5.690,149.252
C01283=1182.281,-89.267,-40.910,179.177,5.689,149.253
C01284=1182.287,-89.516,-40.900,179.175,5.689,149.253
C01285=1182.292,-89.767,-40.889,179.173,5.689,149.254
C01286=1182.297,-90.016,-40.879,179.171,5.688,149.254
C01287=1182.303,-90.266,-40.870,179.169,5.689,149.255
C01288=1182.308,-90.516,-40.860,179.166,5.688,149.255
C01289=1182.313,-90.766,-40.849,179.164,5.688,149.256
C01290=1182.318,-91.015,-40.840,179.162,5.688,149.257
C01291=1182.324,-91.265,-40.829,179.159,5.687,149.257
C01292=1182.329,-91.515,-40.819,179.157,5.687,149.258
C01293=1182.334,-91.764,-40.809,179.155,5.687,149.259
C01294=1182.340,-92.014,-40.800,179.153,5.687,149.259
C01295=1182.345,-92.264,-40.789,179.151,5.686,149.260
C01296=1182.350,-92.514,-40.779,179.149,5.687,149.260
C01297=1182.355,-92.763,-40.769,179.146,5.686,149.261
C01298=1182.361,-93.013,-40.759,179.144,5.685,149.262
C01299=1182.366,-93.262,-40.749,179.142,5.686,149.262
C01300=1182.371,-93.513,-40.740,179.140,5.685,149.263
C01301=1182.376,-93.762,-40.729,179.138,5.685,149.264
C01302=1182.382,-94.012,-40.719,179.135,5.685,149.264
C01303=1182.387,-94.261,-40.710,179.133,5.685,149.265
C01304=1182.392,-94.512,-40.700,179.131,5.685,149.265
C01305=1182.398,-94.762,-40.690,179.128,5.684,149.266
C01306=1182.403,-95.011,-40.680,179.126,5.684,149.267
C01307=1182.408,-95.260,-40.670,179.124,5.683,149.267
C01308=1182.414,-95.511,-40.660,179.122,5.684,149.268
C01309=1182.418,-95.760,-40.650,179.120,5.683,149.268
C01310=1182.424,-96.010,-40.640,179.118,5.684,149.269
C01311=1182.430,-96.260,-40.630,179.115,5.683,149.270
C01312=1182.435,-96.509,-40.621,179.113,5.682,149.270
C01313=1182.440,-96.759,-40.611,179.111,5.683,149.271
C01314=1182.445,-97.009,-40.601,179.109,5.682,149.271
C01315=1182.451,-97.259,-40.591,179.107,5.682,149.272
C01316=1182.456,-97.509,-40.581,179.104,5.682,149.273
C01317=1182.461,-97.758,-40.571,179.102,5.682,149.273
C01318=1182.467,-98.008,-40.562,179.100,5.682,149.274
C01319=1182.472,-98.258,-40.551,179.097,5.681,149.275
C01320=1182.477,-98.507,-40.542,179.095,5.681,149.275
C01321=1182.483,-98.758,-40.532,179.093,5.680,149.276
C01322=1182.488,-99.007,-40.523,179.091,5.681,149.276
C01323=1182.493,-99.256,-40.512,179.089,5.680,149.277
C01324=1182.498,-99.506,-40.504,179.087,5.680,149.278
C01325=1182.503,-99.757,-40.493,179.085,5.680,149.278
C01326=1182.509,-100.006,-40.483,179.083,5.680,149.279
C01327=1182.514,-100.256,-40.474,179.080,5.679,149.279
C01328=1182.520,-100.505,-40.464,179.078,5.679,149.280
C01329=1182.525,-100.755,-40.455,179.076,5.679,149.281
C01330=1182.530,-101.005,-40.445,179.073,5.678,149.281
C01331=1182.535,-101.255,-40.435,179.071,5.679,149.282
C01332=1182.541,-101.526,-40.424,179.069,5.678,149.282
C01333=1182.547,-101.798,-40.414,179.066,5.678,149.283
C01334=1182.552,-102.070,-40.404,179.064,5.678,149.284
C01335=1182.558,-102.341,-40.393,179.062,5.678,149.285
C01336=1182.564,-102.592,-40.383,179.059,5.677,149.285
C01337=1182.568,-102.841,-40.374,179.057,5.677,149.286
C01338=1182.574,-103.091,-40.364,179.055,5.677,149.286
C01339=1182.579,-103.340,-40.354,179.053,5.677,149.287
C01340=1182.585,-103.590,-40.345,179.051,5.676,149.287
C01341=1182.590,-103.840,-40.335,179.049,5.677,149.288
C01342=1182.596,-104.090,-40.326,179.047,5.676,149.289
C01343=1182.600,-104.340,-40.316,179.045,5.676,149.289
C01344=1182.606,-104.590,-40.306,179.042,5.676,149.290
C01345=1182.611,-104.839,-40.297,179.040,5.676,149.291
C01346=1182.617,-105.089,-40.287,179.038,5.675,149.291
C01347=1182.622,-105.339,-40.278,179.036,5.675,149.292
C01348=1182.628,-105.589,-40.268,179.033,5.675,149.292
C01349=1182.632,-105.838,-40.259,179.031,5.674,149.293
C01350=1182.638,-106.088,-40.250,179.029,5.675,149.294
C01351=1182.643,-106.337,-40.239,179.027,5.674,149.294
C01352=1182.648,-106.587,-40.231,179.025,5.674,149.295
C01353=1182.654,-106.837,-40.220,179.023,5.674,149.295
C01354=1182.659,-107.087,-40.211,179.021,5.674,149.296
C01355=1182.664,-107.337,-40.201,179.018,5.673,149.297
C01356=1182.669,-107.587,-40.192,179.016,5.674,149.297
C01357=1182.674,-107.836,-40.183,179.014,5.673,149.298
C01358=1182.680,-108.086,-40.173,179.012,5.673,149.298
C01359=1182.685,-108.336,-40.164,179.010,5.672,149.299
C01360=1182.691,-108.585,-40.154,179.008,5.673,149.300
C01361=1182.696,-108.835,-40.145,179.005,5.672,149.300
C01362=1182.701,-109.085,-40.136,179.003,5.672,149.301
C01363=1182.707,-109.335,-40.126,179.001,5.672,149.301
C01364=1182.712,-109.585,-40.117,178.999,5.671,149.302
C01365=1182.717,-109.834,-40.108,178.997,5.671,149.303
C01366=1182.723,-110.084,-40.098,178.994,5.671,149.303
C01367=1182.728,-110.334,-40.089,178.993,5.671,149.304
C01368=1182.734,-110.584,-40.079,178.990,5.671,149.304
C01369=1182.739,-110.833,-40.070,178.988,5.671,149.305
C01370=1182.744,-111.083,-40.061,178.986,5.670,149.306
C01371=1182.750,-111.333,-40.051,178.984,5.670,149.306
C01372=1182.755,-111.582,-40.042,178.981,5.670,149.307
C01373=1182.760,-111.832,-40.033,178.980,5.670,149.307
C01374=1182.766,-112.082,-40.023,178.977,5.669,149.308
C01375=1182.770,-112.332,-40.014,178.976,5.669,149.309
C01376=1182.776,-112.581,-40.005,178.973,5.669,149.309
C01377=1182.782,-112.832,-39.995,178.971,5.669,149.310
C01378=1182.786,-113.081,-39.986,178.969,5.669,149.310
C01379=1182.792,-113.331,-39.977,178.967,5.669,149.311
C01380=1182.797,-113.581,-39.967,178.964,5.668,149.312
C01381=1182.803,-113.831,-39.958,178.963,5.668,149.312
C01382=1182.807,-114.080,-39.949,178.960,5.668,149.313
C01383=1182.813,-114.330,-39.940,178.958,5.668,149.313
C01384=1182.819,-114.580,-39.930,178.956,5.668,149.314
C01385=1182.824,-114.830,-39.922,178.954,5.668,149.315
C01386=1182.829,-115.080,-39.913,178.951,5.667,149.315
C01387=1182.834,-115.329,-39.902,178.950,5.667,149.316
C01388=1182.840,-115.579,-39.894,178.947,5.667,149.316
C01389=1182.845,-115.829,-39.885,178.946,5.667,149.317
C01390=1182.850,-116.079,-39.876,178.943,5.666,149.318
C01391=1182.856,-116.329,-39.866,178.941,5.667,149.318
C01392=1182.861,-116.578,-39.857,178.939,5.666,149.319
C01393=1182.866,-116.828,-39.848,178.937,5.666,149.319
C01394=1182.871,-117.078,-39.839,178.934,5.666,149.320
C01395=1182.878,-117.327,-39.830,178.933,5.666,149.321
C01396=1182.883,-117.577,-39.821,178.930,5.665,149.321
C01397=1182.888,-117.827,-39.812,178.929,5.665,149.322
C01398=1182.893,-118.076,-39.802,178.926,5.665,149.322
C01399=1182.898,-118.326,-39.793,178.924,5.665,149.323
C01400=1182.904,-118.576,-39.784,178.922,5.665,149.324
C01401=1182.909,-118.826,-39.775,178.920,5.665,149.324
C01402=1182.914,-119.076,-39.766,178.918,5.664,149.325
C01403=1182.919,-119.326,-39.757,178.916,5.664,149.325
C01404=1182.925,-119.576,-39.748,178.913,5.664,149.326
C01405=1182.930,-119.826,-39.739,178.911,5.664,149.327
C01406=1182.935,-120.075,-39.729,178.909,5.663,149.327
C01407=1182.940,-120.325,-39.720,178.907,5.664,149.328
C01408=1182.946,-120.574,-39.712,178.905,5.663,149.328
C01409=1182.951,-120.824,-39.703,178.903,5.663,149.329
C01410=1182.957,-121.074,-39.694,178.901,5.662,149.329
C01411=1182.962,-121.324,-39.685,178.899,5.663,149.330
C01412=1182.968,-121.574,-39.676,178.896,5.662,149.331
C01413=1182.973,-121.824,-39.667,178.894,5.663,149.331
C01414=1182.978,-122.074,-39.658,178.892,5.662,149.332
C01415=1182.983,-122.323,-39.649,178.891,5.662,149.332
C01416=1182.989,-122.573,-39.640,178.888,5.661,149.333
C01417=1182.994,-122.822,-39.631,178.886,5.661,149.334
C01418=1182.999,-123.072,-39.623,178.884,5.661,149.334
C01419=1183.005,-123.322,-39.613,178.882,5.661,149.335
C01420=1183.010,-123.572,-39.604,178.879,5.661,149.335
C01421=1183.015,-123.822,-39.595,178.878,5.661,149.336
C01422=1183.021,-124.072,-39.586,178.875,5.660,149.337
C01423=1183.026,-124.321,-39.578,178.873,5.660,149.337
C01424=1183.032,-124.571,-39.569,178.871,5.660,149.338
C01425=1183.037,-124.821,-39.560,178.869,5.660,149.338
C01426=1183.042,-125.071,-39.551,178.867,5.659,149.339
C01427=1183.047,-125.321,-39.542,178.865,5.660,149.340
C01428=1183.052,-125.570,-39.533,178.863,5.659,149.340
C01429=1183.058,-125.821,-39.524,178.861,5.659,149.341
C01430=1183.064,-126.070,-39.515,178.858,5.659,149.341
C01431=1183.069,-126.320,-39.506,178.857,5.659,149.342
C01432=1183.074,-126.569,-39.498,178.855,5.659,149.342
C01433=1183.079,-126.819,-39.489,178.852,5.658,149.343
C01434=1183.085,-127.069,-39.480,178.850,5.659,149.344
C01435=1183.090,-127.318,-39.471,178.848,5.658,149.344
C01436=1182.669,-127.330,-39.511,178.844,5.661,149.346
C01437=1182.663,-127.080,-39.520,178.846,5.662,149.346
C01438=1182.658,-126.830,-39.529,178.849,5.661,149.345
C01439=1182.653,-126.581,-39.538,178.851,5.662,149.344
C01440=1182.647,-126.331,-39.547,178.852,5.662,149.344
C01441=1182.642,-126.081,-39.555,178.855,5.663,149.343
C01442=1182.637,-125.831,-39.564,178.857,5.663,149.343
C01443=1182.632,-125.581,-39.573,178.859,5.663,149.342
C01444=1182.627,-125.331,-39.582,178.861,5.663,149.341
C01445=1182.621,-125.082,-39.591,178.864,5.663,149.341
C01446=1182.616,-124.832,-39.600,178.865,5.663,149.340
C01447=1182.610,-124.582,-39.609,178.867,5.664,149.340
C01448=1182.605,-124.332,-39.618,178.869,5.664,149.339
C01449=1182.600,-124.083,-39.627,178.871,5.664,149.339
C01450=1182.594,-123.832,-39.635,178.874,5.664,149.338
C01451=1182.588,-123.583,-39.644,178.875,5.664,149.337
C01452=1182.583,-123.333,-39.652,178.878,5.664,149.337
C01453=1182.578,-123.083,-39.661,178.880,5.664,149.336
C01454=1182.573,-122.834,-39.671,178.882,5.665,149.335
C01455=1182.568,-122.584,-39.680,178.884,5.665,149.335
C01456=1182.562,-122.334,-39.689,178.886,5.665,149.334
C01457=1182.557,-122.084,-39.698,178.888,5.665,149.334
C01458=1182.552,-121.834,-39.707,178.890,5.666,149.333
C01459=1182.546,-121.585,-39.716,178.892,5.665,149.333
C01460=1182.541,-121.335,-39.725,178.895,5.666,149.332
C01461=1182.536,-121.085,-39.733,178.897,5.666,149.331
C01462=1182.530,-120.836,-39.742,178.899,5.666,149.331
C01463=1182.524,-120.585,-39.752,178.901,5.666,149.330
C01464=1182.519,-120.336,-39.761,178.903,5.667,149.330
C01465=1182.514,-120.086,-39.770,178.905,5.667,149.329
C01466=1182.509,-119.836,-39.779,178.908,5.667,149.328
C01467=1182.504,-119.586,-39.787,178.909,5.667,149.328
C01468=1182.498,-119.337,-39.796,178.912,5.668,149.327
C01469=1182.492,-119.087,-39.805,178.913,5.668,149.327
C01470=1182.487,-118.837,-39.815,178.916,5.668,149.326
C01471=1182.482,-118.588,-39.824,178.918,5.668,149.326
C01472=1182.477,-118.338,-39.833,178.920,5.668,149.325
C01473=1182.472,-118.088,-39.842,178.922,5.668,149.324
C01474=1182.466,-117.838,-39.851,178.925,5.669,149.324
C01475=1182.461,-117.588,-39.860,178.926,5.669,149.323
C01476=1182.456,-117.338,-39.869,178.929,5.669,149.322
C01477=1182.451,-117.089,-39.879,178.930,5.669,149.322
C01478=1182.446,-116.839,-39.888,178.933,5.669,149.321
C01479=1182.440,-116.589,-39.897,178.935,5.669,149.321
C01480=1182.434,-116.339,-39.906,178.937,5.670,149.320
C01481=1182.429,-116.089,-39.915,178.939,5.670,149.320
C01482=1182.424,-115.840,-39.923,178.941,5.670,149.319
C01483=1182.418,-115.590,-39.934,178.943,5.670,149.318
C01484=1182.413,-115.341,-39.943,178.946,5.671,149.318
C01485=1182.408,-115.091,-39.951,178.948,5.670,149.317
C01486=1182.402,-114.841,-39.961,178.950,5.671,149.317
C01487=1182.397,-114.591,-39.971,178.952,5.671,149.316
C01488=1182.392,-114.341,-39.979,178.954,5.672,149.315
C01489=1182.387,-114.092,-39.988,178.956,5.671,149.315
C01490=1182.381,-113.841,-39.998,178.958,5.672,149.314
C01491=1182.375,-113.592,-40.007,178.960,5.672,149.314
C01492=1182.371,-113.342,-40.016,178.963,5.672,149.313
C01493=1182.365,-113.092,-40.026,178.965,5.672,149.312
C01494=1182.360,-112.842,-40.035,178.967,5.673,149.312
C01495=1182.355,-112.593,-40.044,178.969,5.672,149.311
C01496=1182.349,-112.343,-40.054,178.971,5.673,149.311
C01497=1182.344,-112.093,-40.063,178.973,5.673,149.310
C01498=1182.338,-111.843,-40.072,178.975,5.673,149.309
C01499=1182.334,-111.594,-40.081,178.978,5.674,149.309
C01500=1182.328,-111.344,-40.091,178.980,5.674,149.308
C01501=1182.322,-111.094,-40.100,178.982,5.674,149.308
C01502=1182.317,-110.844,-40.110,178.984,5.674,149.307
C01503=1182.312,-110.595,-40.119,178.987,5.675,149.306
C01504=1182.307,-110.345,-40.128,178.988,5.675,149.306
C01505=1182.301,-110.095,-40.138,178.991,5.675,149.305
C01506=1182.296,-109.845,-40.147,178.993,5.675,149.305
C01507=1182.291,-109.595,-40.156,178.995,5.675,149.304
C01508=1182.285,-109.346,-40.166,178.997,5.675,149.303
C01509=1182.280,-109.096,-40.175,179.000,5.676,149.303
C01510=1182.275,-108.846,-40.184,179.001,5.676,149.302
C01511=1182.269,-108.597,-40.194,179.004,5.676,149.302
C01512=1182.264,-108.347,-40.203,179.005,5.676,149.301
C01513=1182.258,-108.097,-40.213,179.008,5.676,149.300
C01514=1182.253,-107.847,-40.222,179.010,5.676,149.300
C01515=1182.249,-107.597,-40.231,179.012,5.677,149.299
C01516=1182.243,-107.347,-40.241,179.014,5.677,149.299
C01517=1182.238,-107.098,-40.250,179.017,5.677,149.298
C01518=1182.232,-106.848,-40.260,179.019,5.678,149.297
C01519=1182.227,-106.598,-40.269,179.021,5.678,149.297
C01520=1182.221,-106.349,-40.280,179.023,5.678,149.296
C01521=1182.216,-106.099,-40.288,179.025,5.678,149.296
C01522=1182.211,-105.849,-40.297,179.027,5.679,149.295
C01523=1182.206,-105.599,-40.308,179.029,5.678,149.294
C01524=1182.200,-105.349,-40.316,179.032,5.679,149.294
C01525=1182.195,-105.100,-40.327,179.034,5.679,149.293
C01526=1182.190,-104.850,-40.336,179.036,5.679,149.292
C01527=1182.184,-104.601,-40.346,179.038,5.679,149.292
C01528=1182.179,-104.350,-40.355,179.041,5.679,149.291
C01529=1182.174,-104.100,-40.365,179.042,5.679,149.291
C01530=1182.169,-103.851,-40.374,179.045,5.680,149.290
C01531=1182.164,-103.601,-40.384,179.047,5.681,149.290
C01532=1182.158,-103.351,-40.393,179.049,5.680,149.289
C01533=1182.153,-103.102,-40.403,179.051,5.681,149.288
C01534=1182.147,-102.852,-40.412,179.053,5.681,149.288
C01535=1182.142,-102.603,-40.422,179.056,5.681,149.287
C01536=1182.137,-102.352,-40.433,179.058,5.681,149.286
C01537=1182.131,-102.081,-40.442,179.060,5.681,149.286
C01538=1182.126,-101.809,-40.453,179.063,5.682,149.285
C01539=1182.119,-101.537,-40.463,179.065,5.682,149.285
C01540=1182.114,-101.266,-40.474,179.067,5.682,149.284
C01541=1182.108,-101.015,-40.484,179.070,5.683,149.283
C01542=1182.104,-100.766,-40.493,179.072,5.682,149.283
C01543=1182.098,-100.516,-40.503,179.074,5.683,149.282
C01544=1182.093,-100.267,-40.513,179.076,5.683,149.281
C01545=1182.087,-100.017,-40.523,179.079,5.683,149.281
C01546=1182.083,-99.767,-40.532,179.080,5.683,149.280
C01547=1182.077,-99.517,-40.542,179.083,5.684,149.279
C01548=1182.072,-99.267,-40.551,179.084,5.684,149.279
C01549=1182.066,-99.018,-40.561,179.087,5.684,149.278
C01550=1182.061,-98.768,-40.572,179.089,5.685,149.278
C01551=1182.055,-98.518,-40.580,179.091,5.684,149.277
C01552=1182.050,-98.269,-40.591,179.094,5.685,149.277
C01553=1182.046,-98.019,-40.601,179.096,5.685,149.276
C01554=1182.040,-97.769,-40.610,179.098,5.686,149.275
C01555=1182.034,-97.519,-40.620,179.100,5.685,149.275
C01556=1182.029,-97.270,-40.630,179.103,5.686,149.274
C01557=1182.023,-97.020,-40.639,179.104,5.686,149.274
C01558=1182.019,-96.770,-40.649,179.107,5.686,149.273
C01559=1182.013,-96.520,-40.660,179.109,5.687,149.272
C01560=1182.008,-96.271,-40.670,179.111,5.686,149.272
C01561=1182.003,-96.021,-40.679,179.113,5.687,149.271
C01562=1181.997,-95.771,-40.689,179.115,5.687,149.270
C01563=1181.992,-95.521,-40.700,179.118,5.687,149.270
C01564=1181.987,-95.271,-40.708,179.120,5.687,149.269
C01565=1181.981,-95.022,-40.719,179.122,5.687,149.269
C01566=1181.976,-94.773,-40.728,179.125,5.688,149.268
C01567=1181.971,-94.523,-40.738,179.127,5.688,149.267
C01568=1181.966,-94.272,-40.748,179.129,5.689,149.267
C01569=1181.961,-94.023,-40.758,179.131,5.688,149.266
C01570=1181.955,-93.773,-40.768,179.133,5.689,149.266
C01571=1181.950,-93.524,-40.778,179.136,5.689,149.265
C01572=1181.945,-93.274,-40.789,179.138,5.689,149.264
C01573=1181.939,-93.024,-40.798,179.140,5.690,149.264
C01574=1181.934,-92.774,-40.808,179.142,5.689,149.263
C01575=1181.928,-92.525,-40.818,179.144,5.690,149.263
C01576=1181.924,-92.275,-40.828,179.146,5.690,149.262
C01577=1181.918,-92.025,-40.838,179.149,5.691,149.261
C01578=1181.912,-91.775,-40.848,179.151,5.691,149.261
C01579=1181.908,-91.526,-40.858,179.153,5.691,149.260
C01580=1181.903,-91.276,-40.868,179.156,5.691,149.259
C01581=1181.897,-91.026,-40.878,179.158,5.691,149.259
C01582=1181.891,-90.776,-40.889,179.160,5.692,149.258
C01583=1181.887,-90.527,-40.899,179.163,5.692,149.258
C01584=1181.881,-90.277,-40.909,179.164,5.692,149.257
C01585=1181.876,-90.027,-40.918,179.167,5.693,149.256
C01586=1181.870,-89.777,-40.928,179.169,5.692,149.256
C01587=1181.866,-89.527,-40.938,179.171,5.693,149.255
C01588=1181.860,-89.278,-40.949,179.173,5.693,149.254
C01589=1181.855,-89.028,-40.959,179.175,5.693,149.254
C01590=1181.850,-88.778,-40.969,179.178,5.694,149.253
C01591=1181.845,-88.529,-40.979,179.180,5.693,149.253
C01592=1181.839,-88.279,-40.989,179.182,5.694,149.252
C01593=1181.834,-88.029,-41.000,179.184,5.694,149.251
C01594=1181.828,-87.779,-41.010,179.187,5.695,149.251
C01595=1181.823,-87.530,-41.020,179.189,5.695,149.250
C01596=1181.819,-87.280,-41.030,179.191,5.695,149.249
C01597=1181.813,-87.030,-41.040,179.193,5.695,149.249
C01598=1181.807,-86.780,-41.050,179.196,5.695,149.248
C01599=1181.802,-86.530,-41.060,179.198,5.696,149.248
C01600=1181.797,-86.280,-41.071,179.200,5.696,149.247
C01601=1181.792,-86.031,-41.080,179.202,5.696,149.247
C01602=1181.787,-85.781,-41.091,179.205,5.697,149.246
C01603=1181.781,-85.531,-41.101,179.207,5.696,149.245
C01604=1181.775,-85.282,-41.111,179.209,5.697,149.245
C01605=1181.770,-85.032,-41.122,179.212,5.697,149.244
C01606=1181.765,-84.782,-41.132,179.213,5.697,149.243
C01607=1181.760,-84.533,-41.142,179.216,5.698,149.243
C01608=1181.755,-84.283,-41.153,179.218,5.697,149.242
C01609=1181.750,-84.034,-41.163,179.220,5.698,149.242
C01610=1181.744,-83.784,-41.173,179.223,5.699,149.241
C01611=1181.739,-83.534,-41.184,179.224,5.699,149.240
C01612=1181.734,-83.284,-41.194,179.227,5.699,149.240
C01613=1181.729,-83.034,-41.205,179.230,5.699,149.239
C01614=1181.724,-82.785,-41.214,179.231,5.699,149.238
C01615=1181.718,-82.535,-41.225,179.234,5.700,149.238
C01616=1181.713,-82.285,-41.235,179.236,5.700,149.237
C01617=1181.707,-82.036,-41.245,179.238,5.700,149.237
C01618=1181.702,-81.785,-41.256,179.241,5.701,149.236
C01619=1181.697,-81.536,-41.266,179.243,5.701,149.235
C01620=1181.692,-81.287,-41.277,179.245,5.701,149.235
C01621=1181.687,-81.037,-41.288,179.247,5.702,149.234
C01622=1181.681,-80.787,-41.298,179.250,5.701,149.233
C01623=1181.676,-80.537,-41.308,179.252,5.702,149.233
C01624=1181.670,-80.287,-41.319,179.254,5.702,149.232
C01625=1181.665,-80.038,-41.329,179.256,5.702,149.232
C01626=1181.660,-79.788,-41.339,179.259,5.703,149.231
C01627=1181.655,-79.539,-41.350,179.261,5.703,149.230
C01628=1181.650,-79.289,-41.360,179.263,5.703,149.230
C01629=1181.645,-79.039,-41.371,179.266,5.704,149.229
C01630=1181.640,-78.789,-41.381,179.268,5.703,149.229
C01631=1181.634,-78.539,-41.391,179.270,5.704,149.228
C01632=1181.628,-78.290,-41.402,179.272,5.704,149.227
C01633=1181.624,-78.040,-41.413,179.275,5.704,149.227
C01634=1181.618,-77.791,-41.423,179.277,5.705,149.226
C01635=1181.613,-77.540,-41.434,179.279,5.705,149.225
C01636=1181.608,-77.291,-41.444,179.282,5.705,149.225
C01637=1181.603,-77.041,-41.455,179.284,5.706,149.224
C01638=1181.597,-76.792,-41.465,179.286,5.705,149.224
C01639=1181.592,-76.541,-41.476,179.289,5.706,149.223
C01640=1181.587,-76.292,-41.486,179.291,5.707,149.222
C01641=1181.581,-76.021,-41.498,179.293,5.706,149.222
C01642=1181.575,-75.750,-41.509,179.295,5.707,149.221
C01643=1181.570,-75.479,-41.521,179.298,5.707,149.220
C01644=1181.564,-75.208,-41.533,179.301,5.707,149.219
C01645=1181.558,-74.958,-41.543,179.302,5.707,149.219
C01646=1181.553,-74.709,-41.554,179.305,5.708,149.218
C01647=1181.548,-74.459,-41.564,179.307,5.709,149.218
C01648=1181.543,-74.209,-41.575,179.309,5.708,149.217
C01649=1181.538,-73.960,-41.586,179.312,5.709,149.216
C01650=1181.533,-73.710,-41.596,179.314,5.710,149.216
C01651=1181.527,-73.460,-41.607,179.316,5.709,149.215
C01652=1181.522,-73.210,-41.619,179.319,5.710,149.215
C01653=1181.516,-72.961,-41.629,179.321,5.710,149.214
C01654=1181.511,-72.710,-41.639,179.323,5.710,149.213
C01655=1181.506,-72.461,-41.650,179.325,5.711,149.213
C01656=1181.501,-72.211,-41.661,179.327,5.710,149.212
C01657=1181.495,-71.962,-41.671,179.330,5.711,149.211
C01658=1181.490,-71.712,-41.682,179.332,5.712,149.211
C01659=1181.485,-71.462,-41.693,179.334,5.711,149.210
C01660=1181.480,-71.213,-41.704,179.337,5.712,149.210
C01661=1181.474,-70.963,-41.715,179.339,5.712,149.209
C01662=1181.469,-70.713,-41.725,179.341,5.712,149.208
C01663=1181.463,-70.464,-41.736,179.344,5.712,149.208
C01664=1181.458,-70.214,-41.747,179.346,5.713,149.207
C01665=1181.454,-69.964,-41.758,179.348,5.713,149.206
C01666=1181.448,-69.714,-41.768,179.350,5.714,149.206
C01667=1181.443,-69.465,-41.780,179.353,5.714,149.205
C01668=1181.437,-69.215,-41.790,179.355,5.714,149.205
C01669=1181.432,-68.965,-41.802,179.357,5.715,149.204
C01670=1181.427,-68.716,-41.812,179.360,5.715,149.203
C01671=1181.422,-68.466,-41.823,179.362,5.715,149.203
C01672=1181.417,-68.216,-41.834,179.364,5.715,149.202
C01673=1181.411,-67.966,-41.844,179.367,5.716,149.201
C01674=1181.406,-67.716,-41.856,179.369,5.715,149.201
C01675=1181.401,-67.467,-41.867,179.371,5.716,149.200
C01676=1181.396,-67.217,-41.877,179.374,5.717,149.200
C01677=1181.391,-66.968,-41.889,179.376,5.716,149.199
C01678=1181.385,-66.718,-41.899,179.378,5.717,149.198
C01679=1181.380,-66.468,-41.911,179.381,5.717,149.198
C01680=1181.375,-66.219,-41.921,179.382,5.717,149.197
C01681=1181.370,-65.969,-41.932,179.385,5.718,149.197
C01682=1181.364,-65.718,-41.943,179.388,5.718,149.196
C01683=1181.359,-65.469,-41.954,179.390,5.719,149.195
C01684=1181.354,-65.219,-41.965,179.392,5.719,149.195
C01685=1181.349,-64.970,-41.976,179.395,5.719,149.194
C01686=1181.343,-64.720,-41.988,179.397,5.720,149.193
C01687=1181.338,-64.470,-41.998,179.399,5.720,149.193
C01688=1181.333,-64.221,-42.009,179.402,5.720,149.192
C01689=1181.328,-63.971,-42.020,179.404,5.721,149.192
C01690=1181.322,-63.721,-42.032,179.406,5.720,149.191
C01691=1181.317,-63.472,-42.043,179.409,5.721,149.190
C01692=1181.312,-63.222,-42.053,179.411,5.722,149.190
C01693=1181.307,-62.972,-42.064,179.413,5.721,149.189
C01694=1181.301,-62.723,-42.076,179.416,5.722,149.188
C01695=1181.296,-62.473,-42.086,179.418,5.722,149.188
C01696=1181.292,-62.223,-42.098,179.420,5.722,149.187
C01697=1181.286,-61.974,-42.109,179.422,5.722,149.186
C01698=1181.281,-61.724,-42.120,179.425,5.723,149.186
C01699=1181.276,-61.474,-42.131,179.427,5.724,149.185
C01700=1181.270,-61.225,-42.143,179.429,5.723,149.184
C01701=1181.265,-60.975,-42.153,179.432,5.724,149.184
C01702=1181.260,-60.725,-42.165,179.434,5.725,149.183
C01703=1181.254,-60.476,-42.176,179.436,5.725,149.183
C01704=1181.249,-60.225,-42.187,179.439,5.725,149.182
C01705=1181.244,-59.976,-42.198,179.441,5.725,149.181
C01706=1181.238,-59.727,-42.209,179.443,5.725,149.181
C01707=1181.234,-59.477,-42.221,179.445,5.726,149.180
C01708=1181.229,-59.227,-42.231,179.448,5.726,149.180
C01709=1181.223,-58.977,-42.243,179.450,5.727,149.179
C01710=1181.218,-58.728,-42.254,179.452,5.727,149.178
C01711=1181.213,-58.478,-42.266,179.455,5.727,149.178
C01712=1181.208,-58.228,-42.277,179.457,5.728,149.177
C01713=1181.203,-57.978,-42.288,179.459,5.728,149.176
C01714=1181.197,-57.729,-42.299,179.462,5.728,149.176
C01715=1181.192,-57.479,-42.311,179.464,5.729,149.175
C01716=1181.188,-57.230,-42.322,179.467,5.729,149.175
C01717=1181.182,-56.979,-42.333,179.469,5.729,149.174
C01718=1181.176,-56.730,-42.344,179.471,5.730,149.173
C01719=1181.171,-56.480,-42.356,179.474,5.730,149.173
C01720=1181.166,-56.230,-42.367,179.476,5.730,149.172
C01721=1181.161,-55.981,-42.379,179.478,5.731,149.171
C01722=1181.156,-55.732,-42.390,179.481,5.731,149.171
C01723=1181.151,-55.481,-42.401,179.483,5.731,149.170
C01724=1181.145,-55.231,-42.412,179.485,5.731,149.170
C01725=1181.141,-54.982,-42.424,179.488,5.732,149.169
C01726=1181.134,-54.733,-42.435,179.490,5.732,149.168
C01727=1181.130,-54.483,-42.447,179.492,5.733,149.168
C01728=1181.124,-54.233,-42.458,179.495,5.733,149.167
C01729=1181.120,-53.983,-42.470,179.497,5.733,149.166
C01730=1181.114,-53.733,-42.482,179.499,5.734,149.166
C01731=1181.109,-53.485,-42.493,179.501,5.734,149.165
C01732=1181.104,-53.235,-42.504,179.504,5.734,149.164
C01733=1181.099,-52.984,-42.515,179.506,5.735,149.164
C01734=1181.093,-52.734,-42.527,179.509,5.735,149.163
C01735=1181.088,-52.485,-42.538,179.511,5.735,149.163
C01736=1181.082,-52.236,-42.550,179.513,5.736,149.162
C01737=1181.078,-51.986,-42.561,179.516,5.736,149.161
C01738=1181.072,-51.736,-42.573,179.519,5.736,149.161
C01739=1181.068,-51.486,-42.584,179.520,5.736,149.160
C01740=1181.062,-51.236,-42.596,179.523,5.737,149.159
C01741=1181.057,-50.987,-42.607,179.526,5.737,149.159
C01742=1181.051,-50.738,-42.619,179.528,5.738,149.158
C01743=1181.047,-50.488,-42.630,179.530,5.738,149.158
C01744=1181.041,-50.238,-42.642,179.532,5.738,149.157
C01745=1181.036,-49.968,-42.655,179.535,5.739,149.156
C01746=1181.030,-49.697,-42.667,179.538,5.739,149.155
C01747=1181.024,-49.427,-42.680,179.540,5.740,149.155
C01748=1181.019,-49.157,-42.692,179.543,5.740,149.154
C01749=1181.013,-48.907,-42.704,179.545,5.740,149.154
C01750=1181.008,-48.658,-42.716,179.547,5.740,149.153
C01751=1181.003,-48.408,-42.728,179.550,5.741,149.152
C01752=1180.998,-48.158,-42.739,179.552,5.742,149.152
C01753=1180.993,-47.908,-42.751,179.554,5.741,149.151
C01754=1180.987,-47.658,-42.763,179.557,5.742,149.150
C01755=1180.982,-47.409,-42.774,179.559,5.742,149.150
C01756=1180.977,-47.159,-42.785,179.562,5.743,149.149
C01757=1180.972,-46.910,-42.797,179.564,5.743,149.148
C01758=1180.967,-46.660,-42.809,179.566,5.743,149.148
C01759=1180.961,-46.411,-42.821,179.569,5.744,149.147
C01760=1180.957,-46.161,-42.832,179.571,5.744,149.147
C01761=1180.951,-45.911,-42.844,179.573,5.744,149.146
C01762=1180.946,-45.661,-42.856,179.576,5.745,149.145
C01763=1180.941,-45.411,-42.868,179.578,5.745,149.145
C01764=1180.935,-45.162,-42.879,179.580,5.746,149.144
C01765=1180.930,-44.913,-42.892,179.583,5.746,149.144
C01766=1180.925,-44.663,-42.903,179.585,5.746,149.143
C01767=1180.920,-44.413,-42.915,179.587,5.747,149.142
C01768=1180.915,-44.163,-42.927,179.590,5.747,149.142
C01769=1180.910,-43.914,-42.938,179.593,5.748,149.141
C01770=1180.904,-43.664,-42.950,179.594,5.748,149.140
C01771=1180.899,-43.415,-42.962,179.597,5.748,149.140
C01772=1180.894,-43.165,-42.974,179.600,5.749,149.139
C01773=1180.889,-42.915,-42.986,179.602,5.749,149.139
C01774=1180.884,-42.665,-42.998,179.604,5.749,149.138
C01775=1180.879,-42.416,-43.010,179.607,5.749,149.137
C01776=1180.874,-42.166,-43.021,179.609,5.750,149.136
C01777=1180.868,-41.916,-43.033,179.611,5.751,149.136
C01778=1180.863,-41.666,-43.045,179.614,5.751,149.135
C01779=1180.858,-41.417,-43.058,179.616,5.751,149.135
C01780=1180.853,-41.167,-43.069,179.618,5.752,149.134
C01781=1180.847,-40.918,-43.081,179.621,5.752,149.133
C01782=1180.842,-40.669,-43.093,179.624,5.752,149.133
C01783=1180.837,-40.419,-43.105,179.626,5.753,149.132
C01784=1180.832,-40.169,-43.116,179.628,5.753,149.132
C01785=1180.827,-39.919,-43.128,179.631,5.753,149.131
C01786=1180.821,-39.670,-43.141,179.633,5.754,149.130
C01787=1180.816,-39.420,-43.153,179.635,5.755,149.130
C01788=1180.811,-39.170,-43.165,179.638,5.755,149.129
C01789=1180.806,-38.921,-43.177,179.640,5.755,149.129
C01790=1180.801,-38.671,-43.189,179.642,5.756,149.128
C01791=1180.796,-38.422,-43.201,179.645,5.756,149.127
C01792=1180.790,-38.172,-43.213,179.648,5.756,149.126
C01793=1180.785,-37.922,-43.225,179.649,5.756,149.126
C01794=1180.780,-37.673,-43.238,179.652,5.757,149.125
C01795=1180.775,-37.423,-43.249,179.655,5.757,149.125
C01796=1180.770,-37.173,-43.261,179.657,5.758,149.124
C01797=1180.764,-36.924,-43.273,179.659,5.759,149.123
C01798=1180.759,-36.674,-43.285,179.662,5.759,149.123
C01799=1180.754,-36.424,-43.298,179.664,5.759,149.122
C01800=1180.749,-36.174,-43.310,179.666,5.759,149.121
C01801=1180.744,-35.925,-43.323,179.669,5.760,149.121
C01802=1180.738,-35.675,-43.335,179.671,5.761,149.120
C01803=1180.734,-35.426,-43.347,179.674,5.761,149.120
C01804=1180.729,-35.176,-43.358,179.676,5.761,149.119
C01805=1180.723,-34.926,-43.370,179.679,5.761,149.118
C01806=1180.718,-34.676,-43.383,179.681,5.762,149.118
C01807=1180.713,-34.426,-43.395,179.683,5.763,149.117
C01808=1180.708,-34.177,-43.407,179.686,5.763,149.116
C01809=1180.702,-33.927,-43.419,179.688,5.763,149.116
C01810=1180.697,-33.678,-43.432,179.690,5.763,149.115
C01811=1180.692,-33.428,-43.444,179.693,5.764,149.114
C01812=1180.686,-33.179,-43.456,179.695,5.765,149.114
C01813=1180.681,-32.929,-43.469,179.698,5.765,149.113
C01814=1180.677,-32.680,-43.480,179.701,5.766,149.113
C01815=1180.671,-32.430,-43.493,179.702,5.766,149.112
C01816=1180.667,-32.180,-43.505,179.705,5.766,149.111
C01817=1180.662,-31.930,-43.518,179.707,5.766,149.111
C01818=1180.656,-31.680,-43.530,179.710,5.767,149.110
C01819=1180.651,-31.431,-43.542,179.712,5.768,149.110
C01820=1180.646,-31.181,-43.554,179.715,5.768,149.109
C01821=1180.640,-30.932,-43.567,179.717,5.768,149.108
C01822=1180.635,-30.683,-43.579,179.719,5.769,149.108
C01823=1180.630,-30.433,-43.591,179.722,5.769,149.107
C01824=1180.625,-30.183,-43.604,179.725,5.770,149.106
C01825=1180.620,-29.933,-43.617,179.727,5.770,149.106
C01826=1180.615,-29.683,-43.629,179.729,5.771,149.105
C01827=1180.610,-29.434,-43.641,179.731,5.770,149.104
C01828=1180.604,-29.184,-43.653,179.734,5.771,149.104
C01829=1180.599,-28.935,-43.666,179.736,5.772,149.103
C01830=1180.594,-28.685,-43.678,179.739,5.772,149.103
